  MoveL (T3096) to (114.66, 105.74, 4.1) mm, rotated rx 180 ry 0 rz -180 deg; joints [0, 0, 0, 0, 0, 0]
  Call Extruder 0.46589
  MoveL (T3097) to (103.84, 116.55, 4.1) mm, rotated rx 180 ry 0 rz -180 deg; joints [0, 0, 0, 0, 0, 0]
  Call Extruder 0.07441
  MoveL (T3098) to (103.84, 114.11, 4.1) mm, rotated rx 180 ry 0 rz -180 deg; joints [0, 0, 0, 0, 0, 0]
  Set speed (45.0 mm/s)
  Call Extruder -1.6
  MoveL (T3099) to (103.84, 114.11, 4.1) mm, rotated rx 180 ry 0 rz -180 deg; joints [0, 0, 0, 0, 0, 0]
  Set speed (120.0 mm/s)
  MoveL (T3100) to (103.84, 114.11, 4.1) mm, rotated rx 180 ry 0 rz -180 deg; joints [0, 0, 0, 0, 0, 0]
  Call Extruder -0.38
  MoveL (T3101) to (103.84, 115.17, 4.1) mm, rotated rx 180 ry 0 rz -180 deg; joints [0, 0, 0, 0, 0, 0]
  Set speed (45.0 mm/s)
  Call Extruder -0.02
  MoveL (T3102) to (103.84, 115.17, 4.1) mm, rotated rx 180 ry 0 rz -180 deg; joints [0, 0, 0, 0, 0, 0]
  Set speed (150.0 mm/s)
  MoveL (T3103) to (103.84, 115.17, 6.1) mm, rotated rx 180 ry 0 rz -180 deg; joints [0, 0, 0, 0, 0, 0]
  MoveL (T3104) to (118.71, 121.16, 6.1) mm, rotated rx 180 ry 0 rz -180 deg; joints [0, 0, 0, 0, 0, 0]
  MoveL (T3105) to (118.71, 121.16, 4.1) mm, rotated rx 180 ry 0 rz -180 deg; joints [0, 0, 0, 0, 0, 0]
  Set speed (40.0 mm/s)
  Call Extruder 2.0
  MoveL (T3106) to (118.71, 121.16, 4.1) mm, rotated rx 180 ry 0 rz -180 deg; joints [0, 0, 0, 0, 0, 0]
  Set speed (25.4 mm/s)
  MoveL (T3107) to (118.71, 121.16, 4.1) mm, rotated rx 180 ry 0 rz -180 deg; joints [0, 0, 0, 0, 0, 0]
  Call Extruder 0.07441
  MoveL (T3108) to (121.16, 121.16, 4.1) mm, rotated rx 180 ry 0 rz -180 deg; joints [0, 0, 0, 0, 0, 0]
  Call Extruder 0.7458
  MoveL (T3109) to (103.84, 103.84, 4.1) mm, rotated rx 180 ry 0 rz -180 deg; joints [0, 0, 0, 0, 0, 0]
  Call Extruder 0.07705
  MoveL (T3110) to (106.37, 103.84, 4.1) mm, rotated rx 180 ry 0 rz -180 deg; joints [0, 0, 0, 0, 0, 0]
  Call Extruder 0.02939
  MoveL (T3111) to (106.37, 104.81, 4.1) mm, rotated rx 180 ry 0 rz -180 deg; joints [0, 0, 0, 0, 0, 0]
  Call Extruder 0.10898
  MoveL (T3112) to (103.84, 107.34, 4.1) mm, rotated rx 180 ry 0 rz -180 deg; joints [0, 0, 0, 0, 0, 0]
  Call Extruder 0.03385
  MoveL (T3113) to (103.84, 108.45, 4.1) mm, rotated rx 180 ry 0 rz -180 deg; joints [0, 0, 0, 0, 0, 0]
  Call Extruder 0.54738
  MoveL (T3114) to (116.55, 121.16, 4.1) mm, rotated rx 180 ry 0 rz -180 deg; joints [0, 0, 0, 0, 0, 0]
  Call Extruder 0.03385
  MoveL (T3115) to (117.66, 121.16, 4.1) mm, rotated rx 180 ry 0 rz -180 deg; joints [0, 0, 0, 0, 0, 0]
  Call Extruder 0.15054
  MoveL (T3116) to (121.16, 117.66, 4.1) mm, rotated rx 180 ry 0 rz -180 deg; joints [0, 0, 0, 0, 0, 0]
  Call Extruder 0.03385
  MoveL (T3117) to (121.16, 116.55, 4.1) mm, rotated rx 180 ry 0 rz -180 deg; joints [0, 0, 0, 0, 0, 0]
  Call Extruder 0.46589
  MoveL (T3118) to (110.34, 105.74, 4.1) mm, rotated rx 180 ry 0 rz -180 deg; joints [0, 0, 0, 0, 0, 0]
  Call Extruder 0.0088
  MoveL (T3119) to (110.05, 105.74, 4.1) mm, rotated rx 180 ry 0 rz -180 deg; joints [0, 0, 0, 0, 0, 0]
  Call Extruder 0.26747
  MoveL (T3120) to (103.84, 111.94, 4.1) mm, rotated rx 180 ry 0 rz -180 deg; joints [0, 0, 0, 0, 0, 0]
  Call Extruder 0.03385
  MoveL (T3121) to (103.84, 113.06, 4.1) mm, rotated rx 180 ry 0 rz -180 deg; joints [0, 0, 0, 0, 0, 0]
  Call Extruder 0.34896
  MoveL (T3122) to (111.94, 121.16, 4.1) mm, rotated rx 180 ry 0 rz -180 deg; joints [0, 0, 0, 0, 0, 0]
  Call Extruder 0.03385
  MoveL (T3123) to (113.06, 121.16, 4.1) mm, rotated rx 180 ry 0 rz -180 deg; joints [0, 0, 0, 0, 0, 0]
  Call Extruder 0.29316
  MoveL (T3124) to (119.86, 114.35, 4.1) mm, rotated rx 180 ry 0 rz -180 deg; joints [0, 0, 0, 0, 0, 0]
  Call Extruder 0.03946
  MoveL (T3125) to (121.16, 114.35, 4.1) mm, rotated rx 180 ry 0 rz -180 deg; joints [0, 0, 0, 0, 0, 0]
  Call Extruder 0.03495
  MoveL (T3126) to (121.16, 115.5, 4.1) mm, rotated rx 180 ry 0 rz -180 deg; joints [0, 0, 0, 0, 0, 0]
  Set speed (45.0 mm/s)
  Call Extruder -1.6
  MoveL (T3127) to (121.16, 115.5, 4.1) mm, rotated rx 180 ry 0 rz -180 deg; joints [0, 0, 0, 0, 0, 0]
  Set speed (120.0 mm/s)
  MoveL (T3128) to (121.16, 115.5, 4.1) mm, rotated rx 180 ry 0 rz -180 deg; joints [0, 0, 0, 0, 0, 0]
  Call Extruder -0.38
  MoveL (T3129) to (121.16, 114.43, 4.1) mm, rotated rx 180 ry 0 rz -180 deg; joints [0, 0, 0, 0, 0, 0]
  Set speed (45.0 mm/s)
  Call Extruder -0.02
  MoveL (T3130) to (121.16, 114.43, 4.1) mm, rotated rx 180 ry 0 rz -180 deg; joints [0, 0, 0, 0, 0, 0]
  Set speed (150.0 mm/s)
  MoveL (T3131) to (121.16, 114.43, 6.1) mm, rotated rx 180 ry 0 rz -180 deg; joints [0, 0, 0, 0, 0, 0]
  MoveL (T3132) to (104.34, 103.54, 6.1) mm, rotated rx 180 ry 0 rz -180 deg; joints [0, 0, 0, 0, 0, 0]
  MoveL (T3133) to (104.34, 103.54, 4.3) mm, rotated rx 180 ry 0 rz -180 deg; joints [0, 0, 0, 0, 0, 0]
  Set speed (40.0 mm/s)
  Call Extruder 2.0
  MoveL (T3134) to (104.34, 103.54, 4.3) mm, rotated rx 180 ry 0 rz -180 deg; joints [0, 0, 0, 0, 0, 0]
  Set speed (25.0 mm/s)
  MoveL (T3135) to (104.34, 103.54, 4.3) mm, rotated rx 180 ry 0 rz -180 deg; joints [0, 0, 0, 0, 0, 0]
  Call Extruder 0.07466
  MoveL (T3136) to (106.79, 103.54, 4.3) mm, rotated rx 180 ry 0 rz -180 deg; joints [0, 0, 0, 0, 0, 0]
  Call Extruder 0.05763
  MoveL (T3137) to (106.79, 105.43, 4.3) mm, rotated rx 180 ry 0 rz -180 deg; joints [0, 0, 0, 0, 0, 0]
  Call Extruder 0.11303
  MoveL (T3138) to (110.5, 105.43, 4.3) mm, rotated rx 180 ry 0 rz -180 deg; joints [0, 0, 0, 0, 0, 0]
  Call Extruder 0.05763
  MoveL (T3139) to (110.5, 103.54, 4.3) mm, rotated rx 180 ry 0 rz -180 deg; joints [0, 0, 0, 0, 0, 0]
  Call Extruder 0.09685
  MoveL (T3140) to (113.68, 103.54, 4.3) mm, rotated rx 180 ry 0 rz -180 deg; joints [0, 0, 0, 0, 0, 0]
  Call Extruder 0.05763
  MoveL (T3141) to (113.68, 105.43, 4.3) mm, rotated rx 180 ry 0 rz -180 deg; joints [0, 0, 0, 0, 0, 0]
  Call Extruder 0.11722
  MoveL (T3142) to (117.53, 105.43, 4.3) mm, rotated rx 180 ry 0 rz -180 deg; joints [0, 0, 0, 0, 0, 0]
  Call Extruder 0.05763
  MoveL (T3143) to (117.53, 103.54, 4.3) mm, rotated rx 180 ry 0 rz -180 deg; joints [0, 0, 0, 0, 0, 0]
  Call Extruder 0.11984
  MoveL (T3144) to (121.46, 103.54, 4.3) mm, rotated rx 180 ry 0 rz -180 deg; joints [0, 0, 0, 0, 0, 0]
  Call Extruder 0.2055
  MoveL (T3145) to (121.46, 110.28, 4.3) mm, rotated rx 180 ry 0 rz -180 deg; joints [0, 0, 0, 0, 0, 0]
  Call Extruder 0.05923
  MoveL (T3146) to (119.52, 110.28, 4.3) mm, rotated rx 180 ry 0 rz -180 deg; joints [0, 0, 0, 0, 0, 0]
  Call Extruder 0.11452
  MoveL (T3147) to (119.52, 114.04, 4.3) mm, rotated rx 180 ry 0 rz -180 deg; joints [0, 0, 0, 0, 0, 0]
  Call Extruder 0.05928
  MoveL (T3148) to (121.46, 114.04, 4.3) mm, rotated rx 180 ry 0 rz -180 deg; joints [0, 0, 0, 0, 0, 0]
  Call Extruder 0.22594
  MoveL (T3149) to (121.46, 121.46, 4.3) mm, rotated rx 180 ry 0 rz -180 deg; joints [0, 0, 0, 0, 0, 0]
  Call Extruder 0.54596
  MoveL (T3150) to (103.54, 121.46, 4.3) mm, rotated rx 180 ry 0 rz -180 deg; joints [0, 0, 0, 0, 0, 0]
  Call Extruder 0.54596
  MoveL (T3151) to (103.54, 103.54, 4.3) mm, rotated rx 180 ry 0 rz -180 deg; joints [0, 0, 0, 0, 0, 0]
  Call Extruder 0.02254
  MoveL (T3152) to (104.28, 103.54, 4.3) mm, rotated rx 180 ry 0 rz -180 deg; joints [0, 0, 0, 0, 0, 0]
  Set speed (150.0 mm/s)
  MoveL (T3153) to (103.53, 103.13, 4.3) mm, rotated rx 180 ry 0 rz -180 deg; joints [0, 0, 0, 0, 0, 0]
  Set speed (25.0 mm/s)
  MoveL (T3154) to (103.53, 103.13, 4.3) mm, rotated rx 180 ry 0 rz -180 deg; joints [0, 0, 0, 0, 0, 0]
  Call Extruder 0.11164
  MoveL (T3155) to (107.2, 103.13, 4.3) mm, rotated rx 180 ry 0 rz -180 deg; joints [0, 0, 0, 0, 0, 0]
  Call Extruder 0.05763
  MoveL (T3156) to (107.2, 105.02, 4.3) mm, rotated rx 180 ry 0 rz -180 deg; joints [0, 0, 0, 0, 0, 0]
  Call Extruder 0.08823
  MoveL (T3157) to (110.09, 105.02, 4.3) mm, rotated rx 180 ry 0 rz -180 deg; joints [0, 0, 0, 0, 0, 0]
  Call Extruder 0.05763
  MoveL (T3158) to (110.09, 103.13, 4.3) mm, rotated rx 180 ry 0 rz -180 deg; joints [0, 0, 0, 0, 0, 0]
  Call Extruder 0.12167
  MoveL (T3159) to (114.09, 103.13, 4.3) mm, rotated rx 180 ry 0 rz -180 deg; joints [0, 0, 0, 0, 0, 0]
  Call Extruder 0.05763
  MoveL (T3160) to (114.09, 105.02, 4.3) mm, rotated rx 180 ry 0 rz -180 deg; joints [0, 0, 0, 0, 0, 0]
  Call Extruder 0.09242
  MoveL (T3161) to (117.12, 105.02, 4.3) mm, rotated rx 180 ry 0 rz -180 deg; joints [0, 0, 0, 0, 0, 0]
  Call Extruder 0.05763
  MoveL (T3162) to (117.12, 103.13, 4.3) mm, rotated rx 180 ry 0 rz -180 deg; joints [0, 0, 0, 0, 0, 0]
  Call Extruder 0.14463
  MoveL (T3163) to (121.87, 103.13, 4.3) mm, rotated rx 180 ry 0 rz -180 deg; joints [0, 0, 0, 0, 0, 0]
  Call Extruder 0.23031
  MoveL (T3164) to (121.87, 110.69, 4.3) mm, rotated rx 180 ry 0 rz -180 deg; joints [0, 0, 0, 0, 0, 0]
  Call Extruder 0.05924
  MoveL (T3165) to (119.92, 110.69, 4.3) mm, rotated rx 180 ry 0 rz -180 deg; joints [0, 0, 0, 0, 0, 0]
  Call Extruder 0.08971
  MoveL (T3166) to (119.92, 113.64, 4.3) mm, rotated rx 180 ry 0 rz -180 deg; joints [0, 0, 0, 0, 0, 0]
  Call Extruder 0.05927
  MoveL (T3167) to (121.87, 113.64, 4.3) mm, rotated rx 180 ry 0 rz -180 deg; joints [0, 0, 0, 0, 0, 0]
  Call Extruder 0.25074
  MoveL (T3168) to (121.87, 121.87, 4.3) mm, rotated rx 180 ry 0 rz -180 deg; joints [0, 0, 0, 0, 0, 0]
  Call Extruder 0.57077
  MoveL (T3169) to (103.13, 121.87, 4.3) mm, rotated rx 180 ry 0 rz -180 deg; joints [0, 0, 0, 0, 0, 0]
  Call Extruder 0.57077
  MoveL (T3170) to (103.13, 103.13, 4.3) mm, rotated rx 180 ry 0 rz -180 deg; joints [0, 0, 0, 0, 0, 0]
  Call Extruder 0.01036
  MoveL (T3171) to (103.47, 103.13, 4.3) mm, rotated rx 180 ry 0 rz -180 deg; joints [0, 0, 0, 0, 0, 0]
  Set speed (150.0 mm/s)
  MoveL (T3172) to (102.72, 102.81, 4.3) mm, rotated rx 180 ry 0 rz -180 deg; joints [0, 0, 0, 0, 0, 0]
  Set speed (25.0 mm/s)
  MoveL (T3173) to (102.72, 102.81, 4.3) mm, rotated rx 180 ry 0 rz -180 deg; joints [0, 0, 0, 0, 0, 0]
  Call Extruder 0.00259
  MoveL (T3174) to (102.72, 102.72, 4.3) mm, rotated rx 180 ry 0 rz -180 deg; joints [0, 0, 0, 0, 0, 0]
  Call Extruder 0.14862
  MoveL (T3175) to (107.6, 102.72, 4.3) mm, rotated rx 180 ry 0 rz -180 deg; joints [0, 0, 0, 0, 0, 0]
  Call Extruder 0.05763
  MoveL (T3176) to (107.61, 104.62, 4.3) mm, rotated rx 180 ry 0 rz -180 deg; joints [0, 0, 0, 0, 0, 0]
  Call Extruder 0.06342
  MoveL (T3177) to (109.69, 104.62, 4.3) mm, rotated rx 180 ry 0 rz -180 deg; joints [0, 0, 0, 0, 0, 0]
  Call Extruder 0.05763
  MoveL (T3178) to (109.69, 102.72, 4.3) mm, rotated rx 180 ry 0 rz -180 deg; joints [0, 0, 0, 0, 0, 0]
  Call Extruder 0.14648
  MoveL (T3179) to (114.49, 102.72, 4.3) mm, rotated rx 180 ry 0 rz -180 deg; joints [0, 0, 0, 0, 0, 0]
  Call Extruder 0.05763
  MoveL (T3180) to (114.49, 104.62, 4.3) mm, rotated rx 180 ry 0 rz -180 deg; joints [0, 0, 0, 0, 0, 0]
  Call Extruder 0.06761
  MoveL (T3181) to (116.71, 104.62, 4.3) mm, rotated rx 180 ry 0 rz -180 deg; joints [0, 0, 0, 0, 0, 0]
  Call Extruder 0.05763
  MoveL (T3182) to (116.71, 102.72, 4.3) mm, rotated rx 180 ry 0 rz -180 deg; joints [0, 0, 0, 0, 0, 0]
  Call Extruder 0.16943
  MoveL (T3183) to (122.28, 102.72, 4.3) mm, rotated rx 180 ry 0 rz -180 deg; joints [0, 0, 0, 0, 0, 0]
  Call Extruder 0.25512
  MoveL (T3184) to (122.28, 111.1, 4.3) mm, rotated rx 180 ry 0 rz -180 deg; joints [0, 0, 0, 0, 0, 0]
  Call Extruder 0.05924
  MoveL (T3185) to (120.33, 111.1, 4.3) mm, rotated rx 180 ry 0 rz -180 deg; joints [0, 0, 0, 0, 0, 0]
  Call Extruder 0.06491
  MoveL (T3186) to (120.33, 113.23, 4.3) mm, rotated rx 180 ry 0 rz -180 deg; joints [0, 0, 0, 0, 0, 0]
  Call Extruder 0.05927
  MoveL (T3187) to (122.28, 113.23, 4.3) mm, rotated rx 180 ry 0 rz -180 deg; joints [0, 0, 0, 0, 0, 0]
  Call Extruder 0.27554
  MoveL (T3188) to (122.28, 122.28, 4.3) mm, rotated rx 180 ry 0 rz -180 deg; joints [0, 0, 0, 0, 0, 0]
  Call Extruder 0.59557
  MoveL (T3189) to (102.72, 122.28, 4.3) mm, rotated rx 180 ry 0 rz -180 deg; joints [0, 0, 0, 0, 0, 0]
  Call Extruder 0.59115
  MoveL (T3190) to (102.72, 102.87, 4.3) mm, rotated rx 180 ry 0 rz -180 deg; joints [0, 0, 0, 0, 0, 0]
  Set speed (150.0 mm/s)
  MoveL (T3191) to (102.78, 102.75, 4.3) mm, rotated rx 180 ry 0 rz -180 deg; joints [0, 0, 0, 0, 0, 0]
  Set speed (45.0 mm/s)
  Call Extruder -1.6
  MoveL (T3192) to (102.78, 102.75, 4.3) mm, rotated rx 180 ry 0 rz -180 deg; joints [0, 0, 0, 0, 0, 0]
  Set speed (120.0 mm/s)
  MoveL (T3193) to (102.78, 102.75, 4.3) mm, rotated rx 180 ry 0 rz -180 deg; joints [0, 0, 0, 0, 0, 0]
  Call Extruder -0.05166
  MoveL (T3194) to (102.72, 102.72, 4.3) mm, rotated rx 180 ry 0 rz -180 deg; joints [0, 0, 0, 0, 0, 0]
  Call Extruder -0.32834
  MoveL (T3195) to (103.65, 102.72, 4.3) mm, rotated rx 180 ry 0 rz -180 deg; joints [0, 0, 0, 0, 0, 0]
  Set speed (45.0 mm/s)
  Call Extruder -0.02
  MoveL (T3196) to (103.65, 102.72, 4.3) mm, rotated rx 180 ry 0 rz -180 deg; joints [0, 0, 0, 0, 0, 0]
  Set speed (150.0 mm/s)
  MoveL (T3197) to (103.65, 102.72, 6.3) mm, rotated rx 180 ry 0 rz -180 deg; joints [0, 0, 0, 0, 0, 0]
  MoveL (T3198) to (111.05, 103.66, 6.3) mm, rotated rx 180 ry 0 rz -180 deg; joints [0, 0, 0, 0, 0, 0]
  MoveL (T3199) to (111.05, 103.66, 4.3) mm, rotated rx 180 ry 0 rz -180 deg; joints [0, 0, 0, 0, 0, 0]
  Set speed (40.0 mm/s)
  Call Extruder 2.0
  MoveL (T3200) to (111.05, 103.66, 4.3) mm, rotated rx 180 ry 0 rz -180 deg; joints [0, 0, 0, 0, 0, 0]
  Set speed (25.0 mm/s)
  MoveL (T3201) to (111.05, 103.66, 4.3) mm, rotated rx 180 ry 0 rz -180 deg; joints [0, 0, 0, 0, 0, 0]
  Call Extruder 0.00953
  MoveL (T3202) to (111.24, 103.85, 4.3) mm, rotated rx 180 ry 0 rz -180 deg; joints [0, 0, 0, 0, 0, 0]
  Call Extruder 0.0244
  MoveL (T3203) to (111.24, 104.53, 4.3) mm, rotated rx 180 ry 0 rz -180 deg; joints [0, 0, 0, 0, 0, 0]
  Call Extruder 0.02196
  MoveL (T3204) to (110.81, 104.1, 4.3) mm, rotated rx 180 ry 0 rz -180 deg; joints [0, 0, 0, 0, 0, 0]
  Call Extruder 0.0244
  MoveL (T3205) to (110.81, 104.78, 4.3) mm, rotated rx 180 ry 0 rz -180 deg; joints [0, 0, 0, 0, 0, 0]
  Call Extruder 0.02196
  MoveL (T3206) to (111.24, 105.21, 4.3) mm, rotated rx 180 ry 0 rz -180 deg; joints [0, 0, 0, 0, 0, 0]
  Call Extruder 0.00611
  MoveL (T3207) to (111.24, 105.38, 4.3) mm, rotated rx 180 ry 0 rz -180 deg; joints [0, 0, 0, 0, 0, 0]
  Call Extruder 0.00412
  MoveL (T3208) to (111.16, 105.46, 4.3) mm, rotated rx 180 ry 0 rz -180 deg; joints [0, 0, 0, 0, 0, 0]
  Call Extruder 0.01245
  MoveL (T3209) to (110.81, 105.46, 4.3) mm, rotated rx 180 ry 0 rz -180 deg; joints [0, 0, 0, 0, 0, 0]
  Call Extruder 0.00953
  MoveL (T3210) to (110.62, 105.27, 4.3) mm, rotated rx 180 ry 0 rz -180 deg; joints [0, 0, 0, 0, 0, 0]
  Set speed (150.0 mm/s)
  MoveL (T3211) to (110.74, 105.86, 4.3) mm, rotated rx 180 ry 0 rz -180 deg; joints [0, 0, 0, 0, 0, 0]
  Set speed (25.0 mm/s)
  MoveL (T3212) to (110.74, 105.86, 4.3) mm, rotated rx 180 ry 0 rz -180 deg; joints [0, 0, 0, 0, 0, 0]
  Call Extruder 0.01793
  MoveL (T3213) to (111.33, 105.86, 4.3) mm, rotated rx 180 ry 0 rz -180 deg; joints [0, 0, 0, 0, 0, 0]
  Call Extruder 0.01377
  MoveL (T3214) to (111.65, 105.55, 4.3) mm, rotated rx 180 ry 0 rz -180 deg; joints [0, 0, 0, 0, 0, 0]
  Call Extruder 0.0427
  MoveL (T3215) to (111.64, 104.14, 4.3) mm, rotated rx 180 ry 0 rz -180 deg; joints [0, 0, 0, 0, 0, 0]
  Call Extruder 0.0129
  MoveL (T3216) to (111.94, 103.84, 4.3) mm, rotated rx 180 ry 0 rz -180 deg; joints [0, 0, 0, 0, 0, 0]
  Call Extruder 0.01737
  MoveL (T3217) to (112.52, 103.84, 4.3) mm, rotated rx 180 ry 0 rz -180 deg; joints [0, 0, 0, 0, 0, 0]
  Call Extruder 0.05183
  MoveL (T3218) to (112.51, 105.55, 4.3) mm, rotated rx 180 ry 0 rz -180 deg; joints [0, 0, 0, 0, 0, 0]
  Call Extruder 0.00521
  MoveL (T3219) to (112.64, 105.67, 4.3) mm, rotated rx 180 ry 0 rz -180 deg; joints [0, 0, 0, 0, 0, 0]
  Set speed (150.0 mm/s)
  MoveL (T3220) to (112.74, 103.81, 4.3) mm, rotated rx 180 ry 0 rz -180 deg; joints [0, 0, 0, 0, 0, 0]
  Set speed (25.0 mm/s)
  MoveL (T3221) to (112.74, 103.81, 4.3) mm, rotated rx 180 ry 0 rz -180 deg; joints [0, 0, 0, 0, 0, 0]
  Call Extruder 0.03185
  MoveL (T3222) to (113.37, 104.44, 4.3) mm, rotated rx 180 ry 0 rz -180 deg; joints [0, 0, 0, 0, 0, 0]
  Call Extruder 0.02376
  MoveL (T3223) to (113.37, 105.11, 4.3) mm, rotated rx 180 ry 0 rz -180 deg; joints [0, 0, 0, 0, 0, 0]
  Call Extruder 0.02267
  MoveL (T3224) to (112.92, 104.66, 4.3) mm, rotated rx 180 ry 0 rz -180 deg; joints [0, 0, 0, 0, 0, 0]
  Call Extruder 0.02376
  MoveL (T3225) to (112.92, 105.33, 4.3) mm, rotated rx 180 ry 0 rz -180 deg; joints [0, 0, 0, 0, 0, 0]
  Call Extruder 0.01562
  MoveL (T3226) to (113.23, 105.64, 4.3) mm, rotated rx 180 ry 0 rz -180 deg; joints [0, 0, 0, 0, 0, 0]
  Set speed (45.0 mm/s)
  Call Extruder -1.6
  MoveL (T3227) to (113.23, 105.64, 4.3) mm, rotated rx 180 ry 0 rz -180 deg; joints [0, 0, 0, 0, 0, 0]
  Set speed (120.0 mm/s)
  MoveL (T3228) to (113.23, 105.64, 4.3) mm, rotated rx 180 ry 0 rz -180 deg; joints [0, 0, 0, 0, 0, 0]
  Call Extruder -0.15689
  MoveL (T3229) to (112.92, 105.33, 4.3) mm, rotated rx 180 ry 0 rz -180 deg; joints [0, 0, 0, 0, 0, 0]
  Call Extruder -0.22311
  MoveL (T3230) to (112.92, 104.7, 4.3) mm, rotated rx 180 ry 0 rz -180 deg; joints [0, 0, 0, 0, 0, 0]
  Set speed (45.0 mm/s)
  Call Extruder -0.02
  MoveL (T3231) to (112.92, 104.7, 4.3) mm, rotated rx 180 ry 0 rz -180 deg; joints [0, 0, 0, 0, 0, 0]
  Set speed (150.0 mm/s)
  MoveL (T3232) to (112.92, 104.7, 6.3) mm, rotated rx 180 ry 0 rz -180 deg; joints [0, 0, 0, 0, 0, 0]
  MoveL (T3233) to (121.16, 109.07, 6.3) mm, rotated rx 180 ry 0 rz -180 deg; joints [0, 0, 0, 0, 0, 0]
  MoveL (T3234) to (121.16, 109.07, 4.3) mm, rotated rx 180 ry 0 rz -180 deg; joints [0, 0, 0, 0, 0, 0]
  Set speed (40.0 mm/s)
  Call Extruder 2.0
  MoveL (T3235) to (121.16, 109.07, 4.3) mm, rotated rx 180 ry 0 rz -180 deg; joints [0, 0, 0, 0, 0, 0]
  Set speed (25.0 mm/s)
  MoveL (T3236) to (121.16, 109.07, 4.3) mm, rotated rx 180 ry 0 rz -180 deg; joints [0, 0, 0, 0, 0, 0]
  Call Extruder 0.02783
  MoveL (T3237) to (121.16, 109.98, 4.3) mm, rotated rx 180 ry 0 rz -180 deg; joints [0, 0, 0, 0, 0, 0]
  Call Extruder 0.04657
  MoveL (T3238) to (119.63, 109.98, 4.3) mm, rotated rx 180 ry 0 rz -180 deg; joints [0, 0, 0, 0, 0, 0]
  Call Extruder 0.06587
  MoveL (T3239) to (121.16, 108.45, 4.3) mm, rotated rx 180 ry 0 rz -180 deg; joints [0, 0, 0, 0, 0, 0]
  Call Extruder 0.03385
  MoveL (T3240) to (121.16, 107.34, 4.3) mm, rotated rx 180 ry 0 rz -180 deg; joints [0, 0, 0, 0, 0, 0]
  Call Extruder 0.14318
  MoveL (T3241) to (117.83, 104.02, 4.3) mm, rotated rx 180 ry 0 rz -180 deg; joints [0, 0, 0, 0, 0, 0]
  Call Extruder 0.00521
  MoveL (T3242) to (117.83, 103.84, 4.3) mm, rotated rx 180 ry 0 rz -180 deg; joints [0, 0, 0, 0, 0, 0]
  Call Extruder 0.10124
  MoveL (T3243) to (121.16, 103.84, 4.3) mm, rotated rx 180 ry 0 rz -180 deg; joints [0, 0, 0, 0, 0, 0]
  Call Extruder 0.7458
  MoveL (T3244) to (103.84, 121.16, 4.3) mm, rotated rx 180 ry 0 rz -180 deg; joints [0, 0, 0, 0, 0, 0]
  Call Extruder 0.10645
  MoveL (T3245) to (103.84, 117.66, 4.3) mm, rotated rx 180 ry 0 rz -180 deg; joints [0, 0, 0, 0, 0, 0]
  Call Extruder 0.15054
  MoveL (T3246) to (107.34, 121.16, 4.3) mm, rotated rx 180 ry 0 rz -180 deg; joints [0, 0, 0, 0, 0, 0]
  Call Extruder 0.03385
  MoveL (T3247) to (108.45, 121.16, 4.3) mm, rotated rx 180 ry 0 rz -180 deg; joints [0, 0, 0, 0, 0, 0]
  Call Extruder 0.46362
  MoveL (T3248) to (119.21, 110.39, 4.3) mm, rotated rx 180 ry 0 rz -180 deg; joints [0, 0, 0, 0, 0, 0]
  Call Extruder 0.01201
  MoveL (T3249) to (119.21, 110, 4.3) mm, rotated rx 180 ry 0 rz -180 deg; joints [0, 0, 0, 0, 0, 0]
  Call Extruder 0.1837
  MoveL (T3250) to (114.95, 105.74, 4.3) mm, rotated rx 180 ry 0 rz -180 deg; joints [0, 0, 0, 0, 0, 0]
  Call Extruder 0.00881
  MoveL (T3251) to (114.66, 105.74, 4.3) mm, rotated rx 180 ry 0 rz -180 deg; joints [0, 0, 0, 0, 0, 0]
  Call Extruder 0.46588
  MoveL (T3252) to (103.84, 116.55, 4.3) mm, rotated rx 180 ry 0 rz -180 deg; joints [0, 0, 0, 0, 0, 0]
  Call Extruder 0.07441
  MoveL (T3253) to (103.84, 114.11, 4.3) mm, rotated rx 180 ry 0 rz -180 deg; joints [0, 0, 0, 0, 0, 0]
  Set speed (45.0 mm/s)
  Call Extruder -1.6
  MoveL (T3254) to (103.84, 114.11, 4.3) mm, rotated rx 180 ry 0 rz -180 deg; joints [0, 0, 0, 0, 0, 0]
  Set speed (120.0 mm/s)
  MoveL (T3255) to (103.84, 114.11, 4.3) mm, rotated rx 180 ry 0 rz -180 deg; joints [0, 0, 0, 0, 0, 0]
  Call Extruder -0.38
  MoveL (T3256) to (103.84, 115.17, 4.3) mm, rotated rx 180 ry 0 rz -180 deg; joints [0, 0, 0, 0, 0, 0]
  Set speed (45.0 mm/s)
  Call Extruder -0.02
  MoveL (T3257) to (103.84, 115.17, 4.3) mm, rotated rx 180 ry 0 rz -180 deg; joints [0, 0, 0, 0, 0, 0]
  Set speed (150.0 mm/s)
  MoveL (T3258) to (103.84, 115.17, 6.3) mm, rotated rx 180 ry 0 rz -180 deg; joints [0, 0, 0, 0, 0, 0]
  MoveL (T3259) to (118.71, 121.16, 6.3) mm, rotated rx 180 ry 0 rz -180 deg; joints [0, 0, 0, 0, 0, 0]
  MoveL (T3260) to (118.71, 121.16, 4.3) mm, rotated rx 180 ry 0 rz -180 deg; joints [0, 0, 0, 0, 0, 0]
  Set speed (40.0 mm/s)
  Call Extruder 2.0
  MoveL (T3261) to (118.71, 121.16, 4.3) mm, rotated rx 180 ry 0 rz -180 deg; joints [0, 0, 0, 0, 0, 0]
  Set speed (25.0 mm/s)
  MoveL (T3262) to (118.71, 121.16, 4.3) mm, rotated rx 180 ry 0 rz -180 deg; joints [0, 0, 0, 0, 0, 0]
  Call Extruder 0.07441
  MoveL (T3263) to (121.16, 121.16, 4.3) mm, rotated rx 180 ry 0 rz -180 deg; joints [0, 0, 0, 0, 0, 0]
  Call Extruder 0.7458
  MoveL (T3264) to (103.84, 103.84, 4.3) mm, rotated rx 180 ry 0 rz -180 deg; joints [0, 0, 0, 0, 0, 0]
  Call Extruder 0.08043
  MoveL (T3265) to (106.48, 103.84, 4.3) mm, rotated rx 180 ry 0 rz -180 deg; joints [0, 0, 0, 0, 0, 0]
  Call Extruder 0.02601
  MoveL (T3266) to (106.48, 104.7, 4.3) mm, rotated rx 180 ry 0 rz -180 deg; joints [0, 0, 0, 0, 0, 0]
  Call Extruder 0.11376
  MoveL (T3267) to (103.84, 107.34, 4.3) mm, rotated rx 180 ry 0 rz -180 deg; joints [0, 0, 0, 0, 0, 0]
  Call Extruder 0.03385
  MoveL (T3268) to (103.84, 108.45, 4.3) mm, rotated rx 180 ry 0 rz -180 deg; joints [0, 0, 0, 0, 0, 0]
  Call Extruder 0.54738
  MoveL (T3269) to (116.55, 121.16, 4.3) mm, rotated rx 180 ry 0 rz -180 deg; joints [0, 0, 0, 0, 0, 0]
  Call Extruder 0.03385
  MoveL (T3270) to (117.66, 121.16, 4.3) mm, rotated rx 180 ry 0 rz -180 deg; joints [0, 0, 0, 0, 0, 0]
  Call Extruder 0.15054
  MoveL (T3271) to (121.16, 117.66, 4.3) mm, rotated rx 180 ry 0 rz -180 deg; joints [0, 0, 0, 0, 0, 0]
  Call Extruder 0.03385
  MoveL (T3272) to (121.16, 116.55, 4.3) mm, rotated rx 180 ry 0 rz -180 deg; joints [0, 0, 0, 0, 0, 0]
  Call Extruder 0.46588
  MoveL (T3273) to (110.34, 105.74, 4.3) mm, rotated rx 180 ry 0 rz -180 deg; joints [0, 0, 0, 0, 0, 0]
  Call Extruder 0.00881
  MoveL (T3274) to (110.05, 105.74, 4.3) mm, rotated rx 180 ry 0 rz -180 deg; joints [0, 0, 0, 0, 0, 0]
  Call Extruder 0.26746
  MoveL (T3275) to (103.84, 111.94, 4.3) mm, rotated rx 180 ry 0 rz -180 deg; joints [0, 0, 0, 0, 0, 0]
  Call Extruder 0.03385
  MoveL (T3276) to (103.84, 113.06, 4.3) mm, rotated rx 180 ry 0 rz -180 deg; joints [0, 0, 0, 0, 0, 0]
  Call Extruder 0.34896
  MoveL (T3277) to (111.94, 121.16, 4.3) mm, rotated rx 180 ry 0 rz -180 deg; joints [0, 0, 0, 0, 0, 0]
  Call Extruder 0.03385
  MoveL (T3278) to (113.06, 121.16, 4.3) mm, rotated rx 180 ry 0 rz -180 deg; joints [0, 0, 0, 0, 0, 0]
  Call Extruder 0.29326
  MoveL (T3279) to (119.86, 114.35, 4.3) mm, rotated rx 180 ry 0 rz -180 deg; joints [0, 0, 0, 0, 0, 0]
  Call Extruder 0.03939
  MoveL (T3280) to (121.16, 114.35, 4.3) mm, rotated rx 180 ry 0 rz -180 deg; joints [0, 0, 0, 0, 0, 0]
  Call Extruder 0.03502
  MoveL (T3281) to (121.16, 115.5, 4.3) mm, rotated rx 180 ry 0 rz -180 deg; joints [0, 0, 0, 0, 0, 0]
  Set speed (45.0 mm/s)
  Call Extruder -1.6
  MoveL (T3282) to (121.16, 115.5, 4.3) mm, rotated rx 180 ry 0 rz -180 deg; joints [0, 0, 0, 0, 0, 0]
  Set speed (120.0 mm/s)
  MoveL (T3283) to (121.16, 115.5, 4.3) mm, rotated rx 180 ry 0 rz -180 deg; joints [0, 0, 0, 0, 0, 0]
  Call Extruder -0.38
  MoveL (T3284) to (121.16, 114.43, 4.3) mm, rotated rx 180 ry 0 rz -180 deg; joints [0, 0, 0, 0, 0, 0]
  Set speed (45.0 mm/s)
  Call Extruder -0.02
  MoveL (T3285) to (121.16, 114.43, 4.3) mm, rotated rx 180 ry 0 rz -180 deg; joints [0, 0, 0, 0, 0, 0]
  Set speed (150.0 mm/s)
  MoveL (T3286) to (121.16, 114.43, 6.3) mm, rotated rx 180 ry 0 rz -180 deg; joints [0, 0, 0, 0, 0, 0]
  MoveL (T3287) to (104.34, 103.54, 6.3) mm, rotated rx 180 ry 0 rz -180 deg; joints [0, 0, 0, 0, 0, 0]
  MoveL (T3288) to (104.34, 103.54, 4.5) mm, rotated rx 180 ry 0 rz -180 deg; joints [0, 0, 0, 0, 0, 0]
  Set speed (40.0 mm/s)
  Call Extruder 2.0
  MoveL (T3289) to (104.34, 103.54, 4.5) mm, rotated rx 180 ry 0 rz -180 deg; joints [0, 0, 0, 0, 0, 0]
  Set speed (25.4 mm/s)
  MoveL (T3290) to (104.34, 103.54, 4.5) mm, rotated rx 180 ry 0 rz -180 deg; joints [0, 0, 0, 0, 0, 0]
  Call Extruder 0.07804
  MoveL (T3291) to (106.9, 103.54, 4.5) mm, rotated rx 180 ry 0 rz -180 deg; joints [0, 0, 0, 0, 0, 0]
  Call Extruder 0.05764
  MoveL (T3292) to (106.9, 105.43, 4.5) mm, rotated rx 180 ry 0 rz -180 deg; joints [0, 0, 0, 0, 0, 0]
  Call Extruder 0.11326
  MoveL (T3293) to (110.62, 105.43, 4.5) mm, rotated rx 180 ry 0 rz -180 deg; joints [0, 0, 0, 0, 0, 0]
  Call Extruder 0.05764
  MoveL (T3294) to (110.62, 103.54, 4.5) mm, rotated rx 180 ry 0 rz -180 deg; joints [0, 0, 0, 0, 0, 0]
  Call Extruder 0.08953
  MoveL (T3295) to (113.56, 103.54, 4.5) mm, rotated rx 180 ry 0 rz -180 deg; joints [0, 0, 0, 0, 0, 0]
  Call Extruder 0.05764
  MoveL (T3296) to (113.56, 105.43, 4.5) mm, rotated rx 180 ry 0 rz -180 deg; joints [0, 0, 0, 0, 0, 0]
  Call Extruder 0.11708
  MoveL (T3297) to (117.4, 105.43, 4.5) mm, rotated rx 180 ry 0 rz -180 deg; joints [0, 0, 0, 0, 0, 0]
  Call Extruder 0.05764
  MoveL (T3298) to (117.4, 103.54, 4.5) mm, rotated rx 180 ry 0 rz -180 deg; joints [0, 0, 0, 0, 0, 0]
  Call Extruder 0.12369
  MoveL (T3299) to (121.46, 103.54, 4.5) mm, rotated rx 180 ry 0 rz -180 deg; joints [0, 0, 0, 0, 0, 0]
  Call Extruder 0.20544
  MoveL (T3300) to (121.46, 110.28, 4.5) mm, rotated rx 180 ry 0 rz -180 deg; joints [0, 0, 0, 0, 0, 0]
  Call Extruder 0.05922
  MoveL (T3301) to (119.52, 110.28, 4.5) mm, rotated rx 180 ry 0 rz -180 deg; joints [0, 0, 0, 0, 0, 0]
  Call Extruder 0.11452
  MoveL (T3302) to (119.52, 114.04, 4.5) mm, rotated rx 180 ry 0 rz -180 deg; joints [0, 0, 0, 0, 0, 0]
  Call Extruder 0.05927
  MoveL (T3303) to (121.46, 114.04, 4.5) mm, rotated rx 180 ry 0 rz -180 deg; joints [0, 0, 0, 0, 0, 0]
  Call Extruder 0.22601
  MoveL (T3304) to (121.46, 121.46, 4.5) mm, rotated rx 180 ry 0 rz -180 deg; joints [0, 0, 0, 0, 0, 0]
  Call Extruder 0.54596
  MoveL (T3305) to (103.54, 121.46, 4.5) mm, rotated rx 180 ry 0 rz -180 deg; joints [0, 0, 0, 0, 0, 0]
  Call Extruder 0.54596
  MoveL (T3306) to (103.54, 103.54, 4.5) mm, rotated rx 180 ry 0 rz -180 deg; joints [0, 0, 0, 0, 0, 0]
  Call Extruder 0.02254
  MoveL (T3307) to (104.28, 103.54, 4.5) mm, rotated rx 180 ry 0 rz -180 deg; joints [0, 0, 0, 0, 0, 0]
  Set speed (150.0 mm/s)
  MoveL (T3308) to (103.53, 103.13, 4.5) mm, rotated rx 180 ry 0 rz -180 deg; joints [0, 0, 0, 0, 0, 0]
  Set speed (25.4 mm/s)
  MoveL (T3309) to (103.53, 103.13, 4.5) mm, rotated rx 180 ry 0 rz -180 deg; joints [0, 0, 0, 0, 0, 0]
  Call Extruder 0.11502
  MoveL (T3310) to (107.31, 103.13, 4.5) mm, rotated rx 180 ry 0 rz -180 deg; joints [0, 0, 0, 0, 0, 0]
  Call Extruder 0.05764
  MoveL (T3311) to (107.31, 105.02, 4.5) mm, rotated rx 180 ry 0 rz -180 deg; joints [0, 0, 0, 0, 0, 0]
  Call Extruder 0.08845
  MoveL (T3312) to (110.21, 105.02, 4.5) mm, rotated rx 180 ry 0 rz -180 deg; joints [0, 0, 0, 0, 0, 0]
  Call Extruder 0.05764
  MoveL (T3313) to (110.21, 103.13, 4.5) mm, rotated rx 180 ry 0 rz -180 deg; joints [0, 0, 0, 0, 0, 0]
  Call Extruder 0.11435
  MoveL (T3314) to (113.97, 103.13, 4.5) mm, rotated rx 180 ry 0 rz -180 deg; joints [0, 0, 0, 0, 0, 0]
  Call Extruder 0.05764
  MoveL (T3315) to (113.96, 105.02, 4.5) mm, rotated rx 180 ry 0 rz -180 deg; joints [0, 0, 0, 0, 0, 0]
  Call Extruder 0.09228
  MoveL (T3316) to (116.99, 105.02, 4.5) mm, rotated rx 180 ry 0 rz -180 deg; joints [0, 0, 0, 0, 0, 0]
  Call Extruder 0.05764
  MoveL (T3317) to (116.99, 103.13, 4.5) mm, rotated rx 180 ry 0 rz -180 deg; joints [0, 0, 0, 0, 0, 0]
  Call Extruder 0.14848
  MoveL (T3318) to (121.87, 103.13, 4.5) mm, rotated rx 180 ry 0 rz -180 deg; joints [0, 0, 0, 0, 0, 0]
  Call Extruder 0.23025
  MoveL (T3319) to (121.87, 110.69, 4.5) mm, rotated rx 180 ry 0 rz -180 deg; joints [0, 0, 0, 0, 0, 0]
  Call Extruder 0.05923
  MoveL (T3320) to (119.92, 110.69, 4.5) mm, rotated rx 180 ry 0 rz -180 deg; joints [0, 0, 0, 0, 0, 0]
  Call Extruder 0.08971
  MoveL (T3321) to (119.92, 113.63, 4.5) mm, rotated rx 180 ry 0 rz -180 deg; joints [0, 0, 0, 0, 0, 0]
  Call Extruder 0.05927
  MoveL (T3322) to (121.87, 113.64, 4.5) mm, rotated rx 180 ry 0 rz -180 deg; joints [0, 0, 0, 0, 0, 0]
  Call Extruder 0.25081
  MoveL (T3323) to (121.87, 121.87, 4.5) mm, rotated rx 180 ry 0 rz -180 deg; joints [0, 0, 0, 0, 0, 0]
  Call Extruder 0.57077
  MoveL (T3324) to (103.13, 121.87, 4.5) mm, rotated rx 180 ry 0 rz -180 deg; joints [0, 0, 0, 0, 0, 0]
  Call Extruder 0.57077
  MoveL (T3325) to (103.13, 103.13, 4.5) mm, rotated rx 180 ry 0 rz -180 deg; joints [0, 0, 0, 0, 0, 0]
  Call Extruder 0.01036
  MoveL (T3326) to (103.47, 103.13, 4.5) mm, rotated rx 180 ry 0 rz -180 deg; joints [0, 0, 0, 0, 0, 0]
  Set speed (150.0 mm/s)
  MoveL (T3327) to (102.72, 102.81, 4.5) mm, rotated rx 180 ry 0 rz -180 deg; joints [0, 0, 0, 0, 0, 0]
  Set speed (25.0 mm/s)
  MoveL (T3328) to (102.72, 102.81, 4.5) mm, rotated rx 180 ry 0 rz -180 deg; joints [0, 0, 0, 0, 0, 0]
  Call Extruder 0.00259
  MoveL (T3329) to (102.72, 102.72, 4.5) mm, rotated rx 180 ry 0 rz -180 deg; joints [0, 0, 0, 0, 0, 0]
  Call Extruder 0.152
  MoveL (T3330) to (107.72, 102.72, 4.5) mm, rotated rx 180 ry 0 rz -180 deg; joints [0, 0, 0, 0, 0, 0]
  Call Extruder 0.05764
  MoveL (T3331) to (107.72, 104.62, 4.5) mm, rotated rx 180 ry 0 rz -180 deg; joints [0, 0, 0, 0, 0, 0]
  Call Extruder 0.06365
  MoveL (T3332) to (109.81, 104.62, 4.5) mm, rotated rx 180 ry 0 rz -180 deg; joints [0, 0, 0, 0, 0, 0]
  Call Extruder 0.05764
  MoveL (T3333) to (109.8, 102.72, 4.5) mm, rotated rx 180 ry 0 rz -180 deg; joints [0, 0, 0, 0, 0, 0]
  Call Extruder 0.13916
  MoveL (T3334) to (114.37, 102.72, 4.5) mm, rotated rx 180 ry 0 rz -180 deg; joints [0, 0, 0, 0, 0, 0]
  Call Extruder 0.05764
  MoveL (T3335) to (114.37, 104.62, 4.5) mm, rotated rx 180 ry 0 rz -180 deg; joints [0, 0, 0, 0, 0, 0]
  Call Extruder 0.06747
  MoveL (T3336) to (116.59, 104.62, 4.5) mm, rotated rx 180 ry 0 rz -180 deg; joints [0, 0, 0, 0, 0, 0]
  Call Extruder 0.05764
  MoveL (T3337) to (116.59, 102.72, 4.5) mm, rotated rx 180 ry 0 rz -180 deg; joints [0, 0, 0, 0, 0, 0]
  Call Extruder 0.17328
  MoveL (T3338) to (122.28, 102.72, 4.5) mm, rotated rx 180 ry 0 rz -180 deg; joints [0, 0, 0, 0, 0, 0]
  Call Extruder 0.25505
  MoveL (T3339) to (122.28, 111.1, 4.5) mm, rotated rx 180 ry 0 rz -180 deg; joints [0, 0, 0, 0, 0, 0]
  Call Extruder 0.05923
  MoveL (T3340) to (120.33, 111.1, 4.5) mm, rotated rx 180 ry 0 rz -180 deg; joints [0, 0, 0, 0, 0, 0]
  Call Extruder 0.06491
  MoveL (T3341) to (120.33, 113.23, 4.5) mm, rotated rx 180 ry 0 rz -180 deg; joints [0, 0, 0, 0, 0, 0]
  Call Extruder 0.05926
  MoveL (T3342) to (122.28, 113.23, 4.5) mm, rotated rx 180 ry 0 rz -180 deg; joints [0, 0, 0, 0, 0, 0]
  Call Extruder 0.2756
  MoveL (T3343) to (122.28, 122.28, 4.5) mm, rotated rx 180 ry 0 rz -180 deg; joints [0, 0, 0, 0, 0, 0]
  Call Extruder 0.59557
  MoveL (T3344) to (102.72, 122.28, 4.5) mm, rotated rx 180 ry 0 rz -180 deg; joints [0, 0, 0, 0, 0, 0]
  Call Extruder 0.59115
  MoveL (T3345) to (102.72, 102.87, 4.5) mm, rotated rx 180 ry 0 rz -180 deg; joints [0, 0, 0, 0, 0, 0]
  Set speed (150.0 mm/s)
  MoveL (T3346) to (102.78, 102.75, 4.5) mm, rotated rx 180 ry 0 rz -180 deg; joints [0, 0, 0, 0, 0, 0]
  Set speed (45.0 mm/s)
  Call Extruder -1.6
  MoveL (T3347) to (102.78, 102.75, 4.5) mm, rotated rx 180 ry 0 rz -180 deg; joints [0, 0, 0, 0, 0, 0]
  Set speed (120.0 mm/s)
  MoveL (T3348) to (102.78, 102.75, 4.5) mm, rotated rx 180 ry 0 rz -180 deg; joints [0, 0, 0, 0, 0, 0]
  Call Extruder -0.05166
  MoveL (T3349) to (102.72, 102.72, 4.5) mm, rotated rx 180 ry 0 rz -180 deg; joints [0, 0, 0, 0, 0, 0]
  Call Extruder -0.32834
  MoveL (T3350) to (103.65, 102.72, 4.5) mm, rotated rx 180 ry 0 rz -180 deg; joints [0, 0, 0, 0, 0, 0]
  Set speed (45.0 mm/s)
  Call Extruder -0.02
  MoveL (T3351) to (103.65, 102.72, 4.5) mm, rotated rx 180 ry 0 rz -180 deg; joints [0, 0, 0, 0, 0, 0]
  Set speed (150.0 mm/s)
  MoveL (T3352) to (103.65, 102.72, 6.5) mm, rotated rx 180 ry 0 rz -180 deg; joints [0, 0, 0, 0, 0, 0]
  MoveL (T3353) to (111.05, 105.64, 6.5) mm, rotated rx 180 ry 0 rz -180 deg; joints [0, 0, 0, 0, 0, 0]
  MoveL (T3354) to (111.05, 105.64, 4.5) mm, rotated rx 180 ry 0 rz -180 deg; joints [0, 0, 0, 0, 0, 0]
  Set speed (40.0 mm/s)
  Call Extruder 2.0
  MoveL (T3355) to (111.05, 105.64, 4.5) mm, rotated rx 180 ry 0 rz -180 deg; joints [0, 0, 0, 0, 0, 0]
  Set speed (25.4 mm/s)
  MoveL (T3356) to (111.05, 105.64, 4.5) mm, rotated rx 180 ry 0 rz -180 deg; joints [0, 0, 0, 0, 0, 0]
  Call Extruder 0.01539
  MoveL (T3357) to (111.36, 105.33, 4.5) mm, rotated rx 180 ry 0 rz -180 deg; joints [0, 0, 0, 0, 0, 0]
  Call Extruder 0.02341
  MoveL (T3358) to (111.36, 104.67, 4.5) mm, rotated rx 180 ry 0 rz -180 deg; joints [0, 0, 0, 0, 0, 0]
  Call Extruder 0.0215
  MoveL (T3359) to (110.92, 105.1, 4.5) mm, rotated rx 180 ry 0 rz -180 deg; joints [0, 0, 0, 0, 0, 0]
  Call Extruder 0.02341
  MoveL (T3360) to (110.92, 104.44, 4.5) mm, rotated rx 180 ry 0 rz -180 deg; joints [0, 0, 0, 0, 0, 0]
  Call Extruder 0.03062
  MoveL (T3361) to (111.54, 103.82, 4.5) mm, rotated rx 180 ry 0 rz -180 deg; joints [0, 0, 0, 0, 0, 0]
  Set speed (45.0 mm/s)
  Call Extruder -1.6
  MoveL (T3362) to (111.54, 103.82, 4.5) mm, rotated rx 180 ry 0 rz -180 deg; joints [0, 0, 0, 0, 0, 0]
  Set speed (120.0 mm/s)
  MoveL (T3363) to (111.54, 103.82, 4.5) mm, rotated rx 180 ry 0 rz -180 deg; joints [0, 0, 0, 0, 0, 0]
  Call Extruder -0.30984
  MoveL (T3364) to (110.92, 104.44, 4.5) mm, rotated rx 180 ry 0 rz -180 deg; joints [0, 0, 0, 0, 0, 0]
  Call Extruder -0.07016
  MoveL (T3365) to (110.92, 104.63, 4.5) mm, rotated rx 180 ry 0 rz -180 deg; joints [0, 0, 0, 0, 0, 0]
  Set speed (45.0 mm/s)
  Call Extruder -0.02
  MoveL (T3366) to (110.92, 104.63, 4.5) mm, rotated rx 180 ry 0 rz -180 deg; joints [0, 0, 0, 0, 0, 0]
  Set speed (150.0 mm/s)
  MoveL (T3367) to (110.92, 104.63, 6.5) mm, rotated rx 180 ry 0 rz -180 deg; joints [0, 0, 0, 0, 0, 0]
  MoveL (T3368) to (110.97, 105.87, 6.5) mm, rotated rx 180 ry 0 rz -180 deg; joints [0, 0, 0, 0, 0, 0]
  MoveL (T3369) to (110.97, 105.87, 4.5) mm, rotated rx 180 ry 0 rz -180 deg; joints [0, 0, 0, 0, 0, 0]
  Set speed (40.0 mm/s)
  Call Extruder 2.0
  MoveL (T3370) to (110.97, 105.87, 4.5) mm, rotated rx 180 ry 0 rz -180 deg; joints [0, 0, 0, 0, 0, 0]
  Set speed (25.4 mm/s)
  MoveL (T3371) to (110.97, 105.87, 4.5) mm, rotated rx 180 ry 0 rz -180 deg; joints [0, 0, 0, 0, 0, 0]
  Call Extruder 0.01432
  MoveL (T3372) to (111.44, 105.87, 4.5) mm, rotated rx 180 ry 0 rz -180 deg; joints [0, 0, 0, 0, 0, 0]
  Call Extruder 0.01377
  MoveL (T3373) to (111.76, 105.55, 4.5) mm, rotated rx 180 ry 0 rz -180 deg; joints [0, 0, 0, 0, 0, 0]
  Call Extruder 0.04632
  MoveL (T3374) to (111.76, 104.03, 4.5) mm, rotated rx 180 ry 0 rz -180 deg; joints [0, 0, 0, 0, 0, 0]
  Call Extruder 0.0078
  MoveL (T3375) to (111.94, 103.84, 4.5) mm, rotated rx 180 ry 0 rz -180 deg; joints [0, 0, 0, 0, 0, 0]
  Call Extruder 0.01366
  MoveL (T3376) to (112.39, 103.84, 4.5) mm, rotated rx 180 ry 0 rz -180 deg; joints [0, 0, 0, 0, 0, 0]
  Call Extruder 0.05183
  MoveL (T3377) to (112.39, 105.55, 4.5) mm, rotated rx 180 ry 0 rz -180 deg; joints [0, 0, 0, 0, 0, 0]
  Call Extruder 0.00892
  MoveL (T3378) to (112.6, 105.75, 4.5) mm, rotated rx 180 ry 0 rz -180 deg; joints [0, 0, 0, 0, 0, 0]
  Set speed (150.0 mm/s)
  MoveL (T3379) to (113.43, 105.27, 4.5) mm, rotated rx 180 ry 0 rz -180 deg; joints [0, 0, 0, 0, 0, 0]
  Set speed (25.4 mm/s)
  MoveL (T3380) to (113.43, 105.27, 4.5) mm, rotated rx 180 ry 0 rz -180 deg; joints [0, 0, 0, 0, 0, 0]
  Call Extruder 0.00974
  MoveL (T3381) to (113.24, 105.46, 4.5) mm, rotated rx 180 ry 0 rz -180 deg; joints [0, 0, 0, 0, 0, 0]
  Call Extruder 0.01318
  MoveL (T3382) to (112.88, 105.46, 4.5) mm, rotated rx 180 ry 0 rz -180 deg; joints [0, 0, 0, 0, 0, 0]
  Call Extruder 0.00415
  MoveL (T3383) to (112.8, 105.38, 4.5) mm, rotated rx 180 ry 0 rz -180 deg; joints [0, 0, 0, 0, 0, 0]
  Call Extruder 0.00571
  MoveL (T3384) to (112.8, 105.22, 4.5) mm, rotated rx 180 ry 0 rz -180 deg; joints [0, 0, 0, 0, 0, 0]
  Call Extruder 0.02315
  MoveL (T3385) to (113.25, 104.77, 4.5) mm, rotated rx 180 ry 0 rz -180 deg; joints [0, 0, 0, 0, 0, 0]
  Call Extruder 0.02476
  MoveL (T3386) to (113.25, 104.08, 4.5) mm, rotated rx 180 ry 0 rz -180 deg; joints [0, 0, 0, 0, 0, 0]
  Call Extruder 0.02315
  MoveL (T3387) to (112.8, 104.54, 4.5) mm, rotated rx 180 ry 0 rz -180 deg; joints [0, 0, 0, 0, 0, 0]
  Call Extruder 0.02476
  MoveL (T3388) to (112.8, 103.85, 4.5) mm, rotated rx 180 ry 0 rz -180 deg; joints [0, 0, 0, 0, 0, 0]
  Call Extruder 0.00973
  MoveL (T3389) to (112.99, 103.66, 4.5) mm, rotated rx 180 ry 0 rz -180 deg; joints [0, 0, 0, 0, 0, 0]
  Set speed (45.0 mm/s)
  Call Extruder -1.6
  MoveL (T3390) to (112.99, 103.66, 4.5) mm, rotated rx 180 ry 0 rz -180 deg; joints [0, 0, 0, 0, 0, 0]
  Set speed (120.0 mm/s)
  MoveL (T3391) to (112.99, 103.66, 4.5) mm, rotated rx 180 ry 0 rz -180 deg; joints [0, 0, 0, 0, 0, 0]
  Call Extruder -0.09573
  MoveL (T3392) to (112.8, 103.85, 4.5) mm, rotated rx 180 ry 0 rz -180 deg; joints [0, 0, 0, 0, 0, 0]
  Call Extruder -0.24376
  MoveL (T3393) to (112.8, 104.54, 4.5) mm, rotated rx 180 ry 0 rz -180 deg; joints [0, 0, 0, 0, 0, 0]
  Call Extruder -0.0405
  MoveL (T3394) to (112.88, 104.45, 4.5) mm, rotated rx 180 ry 0 rz -180 deg; joints [0, 0, 0, 0, 0, 0]
  Set speed (45.0 mm/s)
  Call Extruder -0.02
  MoveL (T3395) to (112.88, 104.45, 4.5) mm, rotated rx 180 ry 0 rz -180 deg; joints [0, 0, 0, 0, 0, 0]
  Set speed (150.0 mm/s)
  MoveL (T3396) to (112.88, 104.45, 6.5) mm, rotated rx 180 ry 0 rz -180 deg; joints [0, 0, 0, 0, 0, 0]
  MoveL (T3397) to (121.16, 109.06, 6.5) mm, rotated rx 180 ry 0 rz -180 deg; joints [0, 0, 0, 0, 0, 0]
  MoveL (T3398) to (121.16, 109.06, 4.5) mm, rotated rx 180 ry 0 rz -180 deg; joints [0, 0, 0, 0, 0, 0]
  Set speed (40.0 mm/s)
  Call Extruder 2.0
  MoveL (T3399) to (121.16, 109.06, 4.5) mm, rotated rx 180 ry 0 rz -180 deg; joints [0, 0, 0, 0, 0, 0]
  Set speed (25.4 mm/s)
  MoveL (T3400) to (121.16, 109.06, 4.5) mm, rotated rx 180 ry 0 rz -180 deg; joints [0, 0, 0, 0, 0, 0]
  Call Extruder 0.0279
  MoveL (T3401) to (121.16, 109.98, 4.5) mm, rotated rx 180 ry 0 rz -180 deg; joints [0, 0, 0, 0, 0, 0]
  Call Extruder 0.04651
  MoveL (T3402) to (119.63, 109.98, 4.5) mm, rotated rx 180 ry 0 rz -180 deg; joints [0, 0, 0, 0, 0, 0]
  Call Extruder 0.06577
  MoveL (T3403) to (121.16, 108.45, 4.5) mm, rotated rx 180 ry 0 rz -180 deg; joints [0, 0, 0, 0, 0, 0]
  Call Extruder 0.03385
  MoveL (T3404) to (121.16, 107.34, 4.5) mm, rotated rx 180 ry 0 rz -180 deg; joints [0, 0, 0, 0, 0, 0]
  Call Extruder 0.14862
  MoveL (T3405) to (117.71, 103.89, 4.5) mm, rotated rx 180 ry 0 rz -180 deg; joints [0, 0, 0, 0, 0, 0]
  Call Extruder 0.00136
  MoveL (T3406) to (117.71, 103.84, 4.5) mm, rotated rx 180 ry 0 rz -180 deg; joints [0, 0, 0, 0, 0, 0]
  Call Extruder 0.10509
  MoveL (T3407) to (121.16, 103.84, 4.5) mm, rotated rx 180 ry 0 rz -180 deg; joints [0, 0, 0, 0, 0, 0]
  Call Extruder 0.7458
  MoveL (T3408) to (103.84, 121.16, 4.5) mm, rotated rx 180 ry 0 rz -180 deg; joints [0, 0, 0, 0, 0, 0]
  Call Extruder 0.10645
  MoveL (T3409) to (103.84, 117.66, 4.5) mm, rotated rx 180 ry 0 rz -180 deg; joints [0, 0, 0, 0, 0, 0]
  Call Extruder 0.15054
  MoveL (T3410) to (107.34, 121.16, 4.5) mm, rotated rx 180 ry 0 rz -180 deg; joints [0, 0, 0, 0, 0, 0]
  Call Extruder 0.03385
  MoveL (T3411) to (108.45, 121.16, 4.5) mm, rotated rx 180 ry 0 rz -180 deg; joints [0, 0, 0, 0, 0, 0]
  Call Extruder 0.46363
  MoveL (T3412) to (119.21, 110.39, 4.5) mm, rotated rx 180 ry 0 rz -180 deg; joints [0, 0, 0, 0, 0, 0]
  Call Extruder 0.01199
  MoveL (T3413) to (119.21, 110, 4.5) mm, rotated rx 180 ry 0 rz -180 deg; joints [0, 0, 0, 0, 0, 0]
  Call Extruder 0.18371
  MoveL (T3414) to (114.95, 105.74, 4.5) mm, rotated rx 180 ry 0 rz -180 deg; joints [0, 0, 0, 0, 0, 0]
  Call Extruder 0.00882
  MoveL (T3415) to (114.66, 105.74, 4.5) mm, rotated rx 180 ry 0 rz -180 deg; joints [0, 0, 0, 0, 0, 0]
  Call Extruder 0.46587
  MoveL (T3416) to (103.84, 116.55, 4.5) mm, rotated rx 180 ry 0 rz -180 deg; joints [0, 0, 0, 0, 0, 0]
  Call Extruder 0.07441
  MoveL (T3417) to (103.84, 114.11, 4.5) mm, rotated rx 180 ry 0 rz -180 deg; joints [0, 0, 0, 0, 0, 0]
  Set speed (45.0 mm/s)
  Call Extruder -1.6
  MoveL (T3418) to (103.84, 114.11, 4.5) mm, rotated rx 180 ry 0 rz -180 deg; joints [0, 0, 0, 0, 0, 0]
  Set speed (120.0 mm/s)
  MoveL (T3419) to (103.84, 114.11, 4.5) mm, rotated rx 180 ry 0 rz -180 deg; joints [0, 0, 0, 0, 0, 0]
  Call Extruder -0.38
  MoveL (T3420) to (103.84, 115.17, 4.5) mm, rotated rx 180 ry 0 rz -180 deg; joints [0, 0, 0, 0, 0, 0]
  Set speed (45.0 mm/s)
  Call Extruder -0.02
  MoveL (T3421) to (103.84, 115.17, 4.5) mm, rotated rx 180 ry 0 rz -180 deg; joints [0, 0, 0, 0, 0, 0]
  Set speed (150.0 mm/s)
  MoveL (T3422) to (103.84, 115.17, 6.5) mm, rotated rx 180 ry 0 rz -180 deg; joints [0, 0, 0, 0, 0, 0]
  MoveL (T3423) to (118.71, 121.16, 6.5) mm, rotated rx 180 ry 0 rz -180 deg; joints [0, 0, 0, 0, 0, 0]
  MoveL (T3424) to (118.71, 121.16, 4.5) mm, rotated rx 180 ry 0 rz -180 deg; joints [0, 0, 0, 0, 0, 0]
  Set speed (40.0 mm/s)
  Call Extruder 2.0
  MoveL (T3425) to (118.71, 121.16, 4.5) mm, rotated rx 180 ry 0 rz -180 deg; joints [0, 0, 0, 0, 0, 0]
  Set speed (25.4 mm/s)
  MoveL (T3426) to (118.71, 121.16, 4.5) mm, rotated rx 180 ry 0 rz -180 deg; joints [0, 0, 0, 0, 0, 0]
  Call Extruder 0.07441
  MoveL (T3427) to (121.16, 121.16, 4.5) mm, rotated rx 180 ry 0 rz -180 deg; joints [0, 0, 0, 0, 0, 0]
  Call Extruder 0.7458
  MoveL (T3428) to (103.84, 103.84, 4.5) mm, rotated rx 180 ry 0 rz -180 deg; joints [0, 0, 0, 0, 0, 0]
  Call Extruder 0.08381
  MoveL (T3429) to (106.6, 103.84, 4.5) mm, rotated rx 180 ry 0 rz -180 deg; joints [0, 0, 0, 0, 0, 0]
  Call Extruder 0.02263
  MoveL (T3430) to (106.6, 104.59, 4.5) mm, rotated rx 180 ry 0 rz -180 deg; joints [0, 0, 0, 0, 0, 0]
  Call Extruder 0.11854
  MoveL (T3431) to (103.84, 107.34, 4.5) mm, rotated rx 180 ry 0 rz -180 deg; joints [0, 0, 0, 0, 0, 0]
  Call Extruder 0.03385
  MoveL (T3432) to (103.84, 108.45, 4.5) mm, rotated rx 180 ry 0 rz -180 deg; joints [0, 0, 0, 0, 0, 0]
  Call Extruder 0.54738
  MoveL (T3433) to (116.55, 121.16, 4.5) mm, rotated rx 180 ry 0 rz -180 deg; joints [0, 0, 0, 0, 0, 0]
  Call Extruder 0.03385
  MoveL (T3434) to (117.66, 121.16, 4.5) mm, rotated rx 180 ry 0 rz -180 deg; joints [0, 0, 0, 0, 0, 0]
  Call Extruder 0.15054
  MoveL (T3435) to (121.16, 117.66, 4.5) mm, rotated rx 180 ry 0 rz -180 deg; joints [0, 0, 0, 0, 0, 0]
  Call Extruder 0.03385
  MoveL (T3436) to (121.16, 116.55, 4.5) mm, rotated rx 180 ry 0 rz -180 deg; joints [0, 0, 0, 0, 0, 0]
  Call Extruder 0.46587
  MoveL (T3437) to (110.34, 105.74, 4.5) mm, rotated rx 180 ry 0 rz -180 deg; joints [0, 0, 0, 0, 0, 0]
  Call Extruder 0.00882
  MoveL (T3438) to (110.05, 105.74, 4.5) mm, rotated rx 180 ry 0 rz -180 deg; joints [0, 0, 0, 0, 0, 0]
  Call Extruder 0.26745
  MoveL (T3439) to (103.84, 111.94, 4.5) mm, rotated rx 180 ry 0 rz -180 deg; joints [0, 0, 0, 0, 0, 0]
  Call Extruder 0.03385
  MoveL (T3440) to (103.84, 113.06, 4.5) mm, rotated rx 180 ry 0 rz -180 deg; joints [0, 0, 0, 0, 0, 0]
  Call Extruder 0.34896
  MoveL (T3441) to (111.94, 121.16, 4.5) mm, rotated rx 180 ry 0 rz -180 deg; joints [0, 0, 0, 0, 0, 0]
  Call Extruder 0.03385
  MoveL (T3442) to (113.06, 121.16, 4.5) mm, rotated rx 180 ry 0 rz -180 deg; joints [0, 0, 0, 0, 0, 0]
  Call Extruder 0.29335
  MoveL (T3443) to (119.86, 114.35, 4.5) mm, rotated rx 180 ry 0 rz -180 deg; joints [0, 0, 0, 0, 0, 0]
  Call Extruder 0.03933
  MoveL (T3444) to (121.16, 114.35, 4.5) mm, rotated rx 180 ry 0 rz -180 deg; joints [0, 0, 0, 0, 0, 0]
  Call Extruder 0.03508
  MoveL (T3445) to (121.16, 115.5, 4.5) mm, rotated rx 180 ry 0 rz -180 deg; joints [0, 0, 0, 0, 0, 0]
  Set speed (45.0 mm/s)
  Call Extruder -1.6
  MoveL (T3446) to (121.16, 115.5, 4.5) mm, rotated rx 180 ry 0 rz -180 deg; joints [0, 0, 0, 0, 0, 0]
  Set speed (120.0 mm/s)
  MoveL (T3447) to (121.16, 115.5, 4.5) mm, rotated rx 180 ry 0 rz -180 deg; joints [0, 0, 0, 0, 0, 0]
  Call Extruder -0.38
  MoveL (T3448) to (121.16, 114.43, 4.5) mm, rotated rx 180 ry 0 rz -180 deg; joints [0, 0, 0, 0, 0, 0]
  Set speed (45.0 mm/s)
  Call Extruder -0.02
  MoveL (T3449) to (121.16, 114.43, 4.5) mm, rotated rx 180 ry 0 rz -180 deg; joints [0, 0, 0, 0, 0, 0]
  Set speed (150.0 mm/s)
  MoveL (T3450) to (121.16, 114.43, 6.5) mm, rotated rx 180 ry 0 rz -180 deg; joints [0, 0, 0, 0, 0, 0]
  MoveL (T3451) to (104.34, 103.54, 6.5) mm, rotated rx 180 ry 0 rz -180 deg; joints [0, 0, 0, 0, 0, 0]
  MoveL (T3452) to (104.34, 103.54, 4.7) mm, rotated rx 180 ry 0 rz -180 deg; joints [0, 0, 0, 0, 0, 0]
  Set speed (40.0 mm/s)
  Call Extruder 2.0
  MoveL (T3453) to (104.34, 103.54, 4.7) mm, rotated rx 180 ry 0 rz -180 deg; joints [0, 0, 0, 0, 0, 0]
  Set speed (26.7 mm/s)
  MoveL (T3454) to (104.34, 103.54, 4.7) mm, rotated rx 180 ry 0 rz -180 deg; joints [0, 0, 0, 0, 0, 0]
  Call Extruder 0.08142
  MoveL (T3455) to (107.01, 103.54, 4.7) mm, rotated rx 180 ry 0 rz -180 deg; joints [0, 0, 0, 0, 0, 0]
  Call Extruder 0.05764
  MoveL (T3456) to (107.01, 105.43, 4.7) mm, rotated rx 180 ry 0 rz -180 deg; joints [0, 0, 0, 0, 0, 0]
  Call Extruder 0.11348
  MoveL (T3457) to (110.74, 105.43, 4.7) mm, rotated rx 180 ry 0 rz -180 deg; joints [0, 0, 0, 0, 0, 0]
  Call Extruder 0.05764
  MoveL (T3458) to (110.74, 103.54, 4.7) mm, rotated rx 180 ry 0 rz -180 deg; joints [0, 0, 0, 0, 0, 0]
  Call Extruder 0.08221
  MoveL (T3459) to (113.44, 103.54, 4.7) mm, rotated rx 180 ry 0 rz -180 deg; joints [0, 0, 0, 0, 0, 0]
  Call Extruder 0.05764
  MoveL (T3460) to (113.44, 105.43, 4.7) mm, rotated rx 180 ry 0 rz -180 deg; joints [0, 0, 0, 0, 0, 0]
  Call Extruder 0.11694
  MoveL (T3461) to (117.27, 105.43, 4.7) mm, rotated rx 180 ry 0 rz -180 deg; joints [0, 0, 0, 0, 0, 0]
  Call Extruder 0.05764
  MoveL (T3462) to (117.27, 103.54, 4.7) mm, rotated rx 180 ry 0 rz -180 deg; joints [0, 0, 0, 0, 0, 0]
  Call Extruder 0.12754
  MoveL (T3463) to (121.46, 103.54, 4.7) mm, rotated rx 180 ry 0 rz -180 deg; joints [0, 0, 0, 0, 0, 0]
  Call Extruder 0.20537
  MoveL (T3464) to (121.46, 110.28, 4.7) mm, rotated rx 180 ry 0 rz -180 deg; joints [0, 0, 0, 0, 0, 0]
  Call Extruder 0.05921
  MoveL (T3465) to (119.52, 110.28, 4.7) mm, rotated rx 180 ry 0 rz -180 deg; joints [0, 0, 0, 0, 0, 0]
  Call Extruder 0.11452
  MoveL (T3466) to (119.52, 114.04, 4.7) mm, rotated rx 180 ry 0 rz -180 deg; joints [0, 0, 0, 0, 0, 0]
  Call Extruder 0.05926
  MoveL (T3467) to (121.46, 114.04, 4.7) mm, rotated rx 180 ry 0 rz -180 deg; joints [0, 0, 0, 0, 0, 0]
  Call Extruder 0.22608
  MoveL (T3468) to (121.46, 121.46, 4.7) mm, rotated rx 180 ry 0 rz -180 deg; joints [0, 0, 0, 0, 0, 0]
  Call Extruder 0.54596
  MoveL (T3469) to (103.54, 121.46, 4.7) mm, rotated rx 180 ry 0 rz -180 deg; joints [0, 0, 0, 0, 0, 0]
  Call Extruder 0.54596
  MoveL (T3470) to (103.54, 103.54, 4.7) mm, rotated rx 180 ry 0 rz -180 deg; joints [0, 0, 0, 0, 0, 0]
  Call Extruder 0.02254
  MoveL (T3471) to (104.28, 103.54, 4.7) mm, rotated rx 180 ry 0 rz -180 deg; joints [0, 0, 0, 0, 0, 0]
  Set speed (150.0 mm/s)
  MoveL (T3472) to (103.53, 103.13, 4.7) mm, rotated rx 180 ry 0 rz -180 deg; joints [0, 0, 0, 0, 0, 0]
  Set speed (26.7 mm/s)
  MoveL (T3473) to (103.53, 103.13, 4.7) mm, rotated rx 180 ry 0 rz -180 deg; joints [0, 0, 0, 0, 0, 0]
  Call Extruder 0.1184
  MoveL (T3474) to (107.42, 103.13, 4.7) mm, rotated rx 180 ry 0 rz -180 deg; joints [0, 0, 0, 0, 0, 0]
  Call Extruder 0.05764
  MoveL (T3475) to (107.42, 105.02, 4.7) mm, rotated rx 180 ry 0 rz -180 deg; joints [0, 0, 0, 0, 0, 0]
  Call Extruder 0.08868
  MoveL (T3476) to (110.33, 105.02, 4.7) mm, rotated rx 180 ry 0 rz -180 deg; joints [0, 0, 0, 0, 0, 0]
  Call Extruder 0.05764
  MoveL (T3477) to (110.33, 103.13, 4.7) mm, rotated rx 180 ry 0 rz -180 deg; joints [0, 0, 0, 0, 0, 0]
  Call Extruder 0.10702
  MoveL (T3478) to (113.84, 103.13, 4.7) mm, rotated rx 180 ry 0 rz -180 deg; joints [0, 0, 0, 0, 0, 0]
  Call Extruder 0.05764
  MoveL (T3479) to (113.84, 105.02, 4.7) mm, rotated rx 180 ry 0 rz -180 deg; joints [0, 0, 0, 0, 0, 0]
  Call Extruder 0.09214
  MoveL (T3480) to (116.87, 105.02, 4.7) mm, rotated rx 180 ry 0 rz -180 deg; joints [0, 0, 0, 0, 0, 0]
  Call Extruder 0.05764
  MoveL (T3481) to (116.87, 103.13, 4.7) mm, rotated rx 180 ry 0 rz -180 deg; joints [0, 0, 0, 0, 0, 0]
  Call Extruder 0.15234
  MoveL (T3482) to (121.87, 103.13, 4.7) mm, rotated rx 180 ry 0 rz -180 deg; joints [0, 0, 0, 0, 0, 0]
  Call Extruder 0.23018
  MoveL (T3483) to (121.87, 110.69, 4.7) mm, rotated rx 180 ry 0 rz -180 deg; joints [0, 0, 0, 0, 0, 0]
  Call Extruder 0.05922
  MoveL (T3484) to (119.92, 110.69, 4.7) mm, rotated rx 180 ry 0 rz -180 deg; joints [0, 0, 0, 0, 0, 0]
  Call Extruder 0.08971
  MoveL (T3485) to (119.92, 113.63, 4.7) mm, rotated rx 180 ry 0 rz -180 deg; joints [0, 0, 0, 0, 0, 0]
  Call Extruder 0.05926
  MoveL (T3486) to (121.87, 113.63, 4.7) mm, rotated rx 180 ry 0 rz -180 deg; joints [0, 0, 0, 0, 0, 0]
  Call Extruder 0.25087
  MoveL (T3487) to (121.87, 121.87, 4.7) mm, rotated rx 180 ry 0 rz -180 deg; joints [0, 0, 0, 0, 0, 0]
  Call Extruder 0.57077
  MoveL (T3488) to (103.13, 121.87, 4.7) mm, rotated rx 180 ry 0 rz -180 deg; joints [0, 0, 0, 0, 0, 0]
  Call Extruder 0.57077
  MoveL (T3489) to (103.13, 103.13, 4.7) mm, rotated rx 180 ry 0 rz -180 deg; joints [0, 0, 0, 0, 0, 0]
  Call Extruder 0.01036
  MoveL (T3490) to (103.47, 103.13, 4.7) mm, rotated rx 180 ry 0 rz -180 deg; joints [0, 0, 0, 0, 0, 0]
  Set speed (150.0 mm/s)
  MoveL (T3491) to (102.72, 102.81, 4.7) mm, rotated rx 180 ry 0 rz -180 deg; joints [0, 0, 0, 0, 0, 0]
  Set speed (25.0 mm/s)
  MoveL (T3492) to (102.72, 102.81, 4.7) mm, rotated rx 180 ry 0 rz -180 deg; joints [0, 0, 0, 0, 0, 0]
  Call Extruder 0.00259
  MoveL (T3493) to (102.72, 102.72, 4.7) mm, rotated rx 180 ry 0 rz -180 deg; joints [0, 0, 0, 0, 0, 0]
  Call Extruder 0.15539
  MoveL (T3494) to (107.83, 102.72, 4.7) mm, rotated rx 180 ry 0 rz -180 deg; joints [0, 0, 0, 0, 0, 0]
  Call Extruder 0.05764
  MoveL (T3495) to (107.83, 104.62, 4.7) mm, rotated rx 180 ry 0 rz -180 deg; joints [0, 0, 0, 0, 0, 0]
  Call Extruder 0.06388
  MoveL (T3496) to (109.92, 104.62, 4.7) mm, rotated rx 180 ry 0 rz -180 deg; joints [0, 0, 0, 0, 0, 0]
  Call Extruder 0.05764
  MoveL (T3497) to (109.92, 102.72, 4.7) mm, rotated rx 180 ry 0 rz -180 deg; joints [0, 0, 0, 0, 0, 0]
  Call Extruder 0.13184
  MoveL (T3498) to (114.25, 102.72, 4.7) mm, rotated rx 180 ry 0 rz -180 deg; joints [0, 0, 0, 0, 0, 0]
  Call Extruder 0.05764
  MoveL (T3499) to (114.25, 104.62, 4.7) mm, rotated rx 180 ry 0 rz -180 deg; joints [0, 0, 0, 0, 0, 0]
  Call Extruder 0.06733
  MoveL (T3500) to (116.46, 104.62, 4.7) mm, rotated rx 180 ry 0 rz -180 deg; joints [0, 0, 0, 0, 0, 0]
  Call Extruder 0.05764
  MoveL (T3501) to (116.46, 102.72, 4.7) mm, rotated rx 180 ry 0 rz -180 deg; joints [0, 0, 0, 0, 0, 0]
  Call Extruder 0.17713
  MoveL (T3502) to (122.28, 102.72, 4.7) mm, rotated rx 180 ry 0 rz -180 deg; joints [0, 0, 0, 0, 0, 0]
  Call Extruder 0.25499
  MoveL (T3503) to (122.28, 111.09, 4.7) mm, rotated rx 180 ry 0 rz -180 deg; joints [0, 0, 0, 0, 0, 0]
  Call Extruder 0.05922
  MoveL (T3504) to (120.33, 111.09, 4.7) mm, rotated rx 180 ry 0 rz -180 deg; joints [0, 0, 0, 0, 0, 0]
  Call Extruder 0.06491
  MoveL (T3505) to (120.33, 113.22, 4.7) mm, rotated rx 180 ry 0 rz -180 deg; joints [0, 0, 0, 0, 0, 0]
  Call Extruder 0.05925
  MoveL (T3506) to (122.28, 113.23, 4.7) mm, rotated rx 180 ry 0 rz -180 deg; joints [0, 0, 0, 0, 0, 0]
  Call Extruder 0.27567
  MoveL (T3507) to (122.28, 122.28, 4.7) mm, rotated rx 180 ry 0 rz -180 deg; joints [0, 0, 0, 0, 0, 0]
  Call Extruder 0.59557
  MoveL (T3508) to (102.72, 122.28, 4.7) mm, rotated rx 180 ry 0 rz -180 deg; joints [0, 0, 0, 0, 0, 0]
  Call Extruder 0.59115
  MoveL (T3509) to (102.72, 102.87, 4.7) mm, rotated rx 180 ry 0 rz -180 deg; joints [0, 0, 0, 0, 0, 0]
  Set speed (150.0 mm/s)
  MoveL (T3510) to (102.78, 102.75, 4.7) mm, rotated rx 180 ry 0 rz -180 deg; joints [0, 0, 0, 0, 0, 0]
  Set speed (45.0 mm/s)
  Call Extruder -1.6
  MoveL (T3511) to (102.78, 102.75, 4.7) mm, rotated rx 180 ry 0 rz -180 deg; joints [0, 0, 0, 0, 0, 0]
  Set speed (120.0 mm/s)
  MoveL (T3512) to (102.78, 102.75, 4.7) mm, rotated rx 180 ry 0 rz -180 deg; joints [0, 0, 0, 0, 0, 0]
  Call Extruder -0.05166
  MoveL (T3513) to (102.72, 102.72, 4.7) mm, rotated rx 180 ry 0 rz -180 deg; joints [0, 0, 0, 0, 0, 0]
  Call Extruder -0.32834
  MoveL (T3514) to (103.65, 102.72, 4.7) mm, rotated rx 180 ry 0 rz -180 deg; joints [0, 0, 0, 0, 0, 0]
  Set speed (45.0 mm/s)
  Call Extruder -0.02
  MoveL (T3515) to (103.65, 102.72, 4.7) mm, rotated rx 180 ry 0 rz -180 deg; joints [0, 0, 0, 0, 0, 0]
  Set speed (150.0 mm/s)
  MoveL (T3516) to (103.65, 102.72, 6.7) mm, rotated rx 180 ry 0 rz -180 deg; joints [0, 0, 0, 0, 0, 0]
  MoveL (T3517) to (106.36, 103.99, 6.7) mm, rotated rx 180 ry 0 rz -180 deg; joints [0, 0, 0, 0, 0, 0]
  MoveL (T3518) to (106.36, 103.99, 4.7) mm, rotated rx 180 ry 0 rz -180 deg; joints [0, 0, 0, 0, 0, 0]
  Set speed (40.0 mm/s)
  Call Extruder 2.0
  MoveL (T3519) to (106.36, 103.99, 4.7) mm, rotated rx 180 ry 0 rz -180 deg; joints [0, 0, 0, 0, 0, 0]
  Set speed (26.7 mm/s)
  MoveL (T3520) to (106.36, 103.99, 4.7) mm, rotated rx 180 ry 0 rz -180 deg; joints [0, 0, 0, 0, 0, 0]
  Call Extruder 0.0156
  MoveL (T3521) to (106.71, 104.33, 4.7) mm, rotated rx 180 ry 0 rz -180 deg; joints [0, 0, 0, 0, 0, 0]
  Call Extruder 0.01892
  MoveL (T3522) to (106.71, 104.93, 4.7) mm, rotated rx 180 ry 0 rz -180 deg; joints [0, 0, 0, 0, 0, 0]
  Call Extruder 0.0074
  MoveL (T3523) to (106.54, 104.77, 4.7) mm, rotated rx 180 ry 0 rz -180 deg; joints [0, 0, 0, 0, 0, 0]
  Call Extruder 0.01892
  MoveL (T3524) to (106.54, 105.36, 4.7) mm, rotated rx 180 ry 0 rz -180 deg; joints [0, 0, 0, 0, 0, 0]
  Call Extruder 0.01231
  MoveL (T3525) to (106.82, 105.64, 4.7) mm, rotated rx 180 ry 0 rz -180 deg; joints [0, 0, 0, 0, 0, 0]
  Set speed (45.0 mm/s)
  Call Extruder -1.6
  MoveL (T3526) to (106.82, 105.64, 4.7) mm, rotated rx 180 ry 0 rz -180 deg; joints [0, 0, 0, 0, 0, 0]
  Set speed (120.0 mm/s)
  MoveL (T3527) to (106.82, 105.64, 4.7) mm, rotated rx 180 ry 0 rz -180 deg; joints [0, 0, 0, 0, 0, 0]
  Call Extruder -0.13863
  MoveL (T3528) to (106.54, 105.36, 4.7) mm, rotated rx 180 ry 0 rz -180 deg; joints [0, 0, 0, 0, 0, 0]
  Call Extruder -0.21308
  MoveL (T3529) to (106.54, 104.77, 4.7) mm, rotated rx 180 ry 0 rz -180 deg; joints [0, 0, 0, 0, 0, 0]
  Call Extruder -0.02829
  MoveL (T3530) to (106.6, 104.82, 4.7) mm, rotated rx 180 ry 0 rz -180 deg; joints [0, 0, 0, 0, 0, 0]
  Set speed (45.0 mm/s)
  Call Extruder -0.02
  MoveL (T3531) to (106.6, 104.82, 4.7) mm, rotated rx 180 ry 0 rz -180 deg; joints [0, 0, 0, 0, 0, 0]
  Set speed (150.0 mm/s)
  MoveL (T3532) to (106.6, 104.82, 6.7) mm, rotated rx 180 ry 0 rz -180 deg; joints [0, 0, 0, 0, 0, 0]
  MoveL (T3533) to (111.21, 105.87, 6.7) mm, rotated rx 180 ry 0 rz -180 deg; joints [0, 0, 0, 0, 0, 0]
  MoveL (T3534) to (111.21, 105.87, 4.7) mm, rotated rx 180 ry 0 rz -180 deg; joints [0, 0, 0, 0, 0, 0]
  Set speed (40.0 mm/s)
  Call Extruder 2.0
  MoveL (T3535) to (111.21, 105.87, 4.7) mm, rotated rx 180 ry 0 rz -180 deg; joints [0, 0, 0, 0, 0, 0]
  Set speed (26.7 mm/s)
  MoveL (T3536) to (111.21, 105.87, 4.7) mm, rotated rx 180 ry 0 rz -180 deg; joints [0, 0, 0, 0, 0, 0]
  Call Extruder 0.01071
  MoveL (T3537) to (111.56, 105.87, 4.7) mm, rotated rx 180 ry 0 rz -180 deg; joints [0, 0, 0, 0, 0, 0]
  Call Extruder 0.01377
  MoveL (T3538) to (111.88, 105.55, 4.7) mm, rotated rx 180 ry 0 rz -180 deg; joints [0, 0, 0, 0, 0, 0]
  Call Extruder 0.04993
  MoveL (T3539) to (111.88, 103.91, 4.7) mm, rotated rx 180 ry 0 rz -180 deg; joints [0, 0, 0, 0, 0, 0]
  Call Extruder 0.0027
  MoveL (T3540) to (111.94, 103.84, 4.7) mm, rotated rx 180 ry 0 rz -180 deg; joints [0, 0, 0, 0, 0, 0]
  Call Extruder 0.00995
  MoveL (T3541) to (112.27, 103.84, 4.7) mm, rotated rx 180 ry 0 rz -180 deg; joints [0, 0, 0, 0, 0, 0]
  Call Extruder 0.05184
  MoveL (T3542) to (112.27, 105.55, 4.7) mm, rotated rx 180 ry 0 rz -180 deg; joints [0, 0, 0, 0, 0, 0]
  Call Extruder 0.01262
  MoveL (T3543) to (112.56, 105.84, 4.7) mm, rotated rx 180 ry 0 rz -180 deg; joints [0, 0, 0, 0, 0, 0]
  Set speed (45.0 mm/s)
  Call Extruder -1.6
  MoveL (T3544) to (112.56, 105.84, 4.7) mm, rotated rx 180 ry 0 rz -180 deg; joints [0, 0, 0, 0, 0, 0]
  Set speed (120.0 mm/s)
  MoveL (T3545) to (112.56, 105.84, 4.7) mm, rotated rx 180 ry 0 rz -180 deg; joints [0, 0, 0, 0, 0, 0]
  Call Extruder -0.14761
  MoveL (T3546) to (112.27, 105.55, 4.7) mm, rotated rx 180 ry 0 rz -180 deg; joints [0, 0, 0, 0, 0, 0]
  Call Extruder -0.23239
  MoveL (T3547) to (112.27, 104.89, 4.7) mm, rotated rx 180 ry 0 rz -180 deg; joints [0, 0, 0, 0, 0, 0]
  Set speed (45.0 mm/s)
  Call Extruder -0.02
  MoveL (T3548) to (112.27, 104.89, 4.7) mm, rotated rx 180 ry 0 rz -180 deg; joints [0, 0, 0, 0, 0, 0]
  Set speed (150.0 mm/s)
  MoveL (T3549) to (112.27, 104.89, 6.7) mm, rotated rx 180 ry 0 rz -180 deg; joints [0, 0, 0, 0, 0, 0]
  MoveL (T3550) to (112.5, 103.81, 6.7) mm, rotated rx 180 ry 0 rz -180 deg; joints [0, 0, 0, 0, 0, 0]
  MoveL (T3551) to (112.5, 103.81, 4.7) mm, rotated rx 180 ry 0 rz -180 deg; joints [0, 0, 0, 0, 0, 0]
  Set speed (40.0 mm/s)
  Call Extruder 2.0
  MoveL (T3552) to (112.5, 103.81, 4.7) mm, rotated rx 180 ry 0 rz -180 deg; joints [0, 0, 0, 0, 0, 0]
  Set speed (26.7 mm/s)
  MoveL (T3553) to (112.5, 103.81, 4.7) mm, rotated rx 180 ry 0 rz -180 deg; joints [0, 0, 0, 0, 0, 0]
  Call Extruder 0.03186
  MoveL (T3554) to (113.13, 104.44, 4.7) mm, rotated rx 180 ry 0 rz -180 deg; joints [0, 0, 0, 0, 0, 0]
  Call Extruder 0.02376
  MoveL (T3555) to (113.13, 105.11, 4.7) mm, rotated rx 180 ry 0 rz -180 deg; joints [0, 0, 0, 0, 0, 0]
  Call Extruder 0.02267
  MoveL (T3556) to (112.68, 104.66, 4.7) mm, rotated rx 180 ry 0 rz -180 deg; joints [0, 0, 0, 0, 0, 0]
  Call Extruder 0.02376
  MoveL (T3557) to (112.68, 105.33, 4.7) mm, rotated rx 180 ry 0 rz -180 deg; joints [0, 0, 0, 0, 0, 0]
  Call Extruder 0.01562
  MoveL (T3558) to (112.99, 105.64, 4.7) mm, rotated rx 180 ry 0 rz -180 deg; joints [0, 0, 0, 0, 0, 0]
  Set speed (45.0 mm/s)
  Call Extruder -1.6
  MoveL (T3559) to (112.99, 105.64, 4.7) mm, rotated rx 180 ry 0 rz -180 deg; joints [0, 0, 0, 0, 0, 0]
  Set speed (120.0 mm/s)
  MoveL (T3560) to (112.99, 105.64, 4.7) mm, rotated rx 180 ry 0 rz -180 deg; joints [0, 0, 0, 0, 0, 0]
  Call Extruder -0.15692
  MoveL (T3561) to (112.68, 105.33, 4.7) mm, rotated rx 180 ry 0 rz -180 deg; joints [0, 0, 0, 0, 0, 0]
  Call Extruder -0.22308
  MoveL (T3562) to (112.68, 104.7, 4.7) mm, rotated rx 180 ry 0 rz -180 deg; joints [0, 0, 0, 0, 0, 0]
  Set speed (45.0 mm/s)
  Call Extruder -0.02
  MoveL (T3563) to (112.68, 104.7, 4.7) mm, rotated rx 180 ry 0 rz -180 deg; joints [0, 0, 0, 0, 0, 0]
  Set speed (150.0 mm/s)
  MoveL (T3564) to (112.68, 104.7, 6.7) mm, rotated rx 180 ry 0 rz -180 deg; joints [0, 0, 0, 0, 0, 0]
  MoveL (T3565) to (111.29, 103.66, 6.7) mm, rotated rx 180 ry 0 rz -180 deg; joints [0, 0, 0, 0, 0, 0]
  MoveL (T3566) to (111.29, 103.66, 4.7) mm, rotated rx 180 ry 0 rz -180 deg; joints [0, 0, 0, 0, 0, 0]
  Set speed (40.0 mm/s)
  Call Extruder 2.0
  MoveL (T3567) to (111.29, 103.66, 4.7) mm, rotated rx 180 ry 0 rz -180 deg; joints [0, 0, 0, 0, 0, 0]
  Set speed (26.7 mm/s)
  MoveL (T3568) to (111.29, 103.66, 4.7) mm, rotated rx 180 ry 0 rz -180 deg; joints [0, 0, 0, 0, 0, 0]
  Call Extruder 0.00954
  MoveL (T3569) to (111.47, 103.85, 4.7) mm, rotated rx 180 ry 0 rz -180 deg; joints [0, 0, 0, 0, 0, 0]
  Call Extruder 0.0244
  MoveL (T3570) to (111.47, 104.53, 4.7) mm, rotated rx 180 ry 0 rz -180 deg; joints [0, 0, 0, 0, 0, 0]
  Call Extruder 0.02197
  MoveL (T3571) to (111.04, 104.1, 4.7) mm, rotated rx 180 ry 0 rz -180 deg; joints [0, 0, 0, 0, 0, 0]
  Call Extruder 0.0244
  MoveL (T3572) to (111.04, 104.78, 4.7) mm, rotated rx 180 ry 0 rz -180 deg; joints [0, 0, 0, 0, 0, 0]
  Call Extruder 0.02197
  MoveL (T3573) to (111.47, 105.21, 4.7) mm, rotated rx 180 ry 0 rz -180 deg; joints [0, 0, 0, 0, 0, 0]
  Call Extruder 0.00611
  MoveL (T3574) to (111.47, 105.38, 4.7) mm, rotated rx 180 ry 0 rz -180 deg; joints [0, 0, 0, 0, 0, 0]
  Call Extruder 0.00412
  MoveL (T3575) to (111.39, 105.46, 4.7) mm, rotated rx 180 ry 0 rz -180 deg; joints [0, 0, 0, 0, 0, 0]
  Call Extruder 0.01245
  MoveL (T3576) to (111.05, 105.46, 4.7) mm, rotated rx 180 ry 0 rz -180 deg; joints [0, 0, 0, 0, 0, 0]
  Call Extruder 0.00953
  MoveL (T3577) to (110.86, 105.27, 4.7) mm, rotated rx 180 ry 0 rz -180 deg; joints [0, 0, 0, 0, 0, 0]
  Set speed (45.0 mm/s)
  Call Extruder -1.6
  MoveL (T3578) to (110.86, 105.27, 4.7) mm, rotated rx 180 ry 0 rz -180 deg; joints [0, 0, 0, 0, 0, 0]
  Set speed (120.0 mm/s)
  MoveL (T3579) to (110.86, 105.27, 4.7) mm, rotated rx 180 ry 0 rz -180 deg; joints [0, 0, 0, 0, 0, 0]
  Call Extruder -0.09452
  MoveL (T3580) to (111.05, 105.46, 4.7) mm, rotated rx 180 ry 0 rz -180 deg; joints [0, 0, 0, 0, 0, 0]
  Call Extruder -0.1235
  MoveL (T3581) to (111.39, 105.46, 4.7) mm, rotated rx 180 ry 0 rz -180 deg; joints [0, 0, 0, 0, 0, 0]
  Call Extruder -0.04086
  MoveL (T3582) to (111.47, 105.38, 4.7) mm, rotated rx 180 ry 0 rz -180 deg; joints [0, 0, 0, 0, 0, 0]
  Call Extruder -0.06061
  MoveL (T3583) to (111.47, 105.21, 4.7) mm, rotated rx 180 ry 0 rz -180 deg; joints [0, 0, 0, 0, 0, 0]
  Call Extruder -0.06051
  MoveL (T3584) to (111.36, 105.09, 4.7) mm, rotated rx 180 ry 0 rz -180 deg; joints [0, 0, 0, 0, 0, 0]
  Set speed (45.0 mm/s)
  Call Extruder -0.02
  MoveL (T3585) to (111.36, 105.09, 4.7) mm, rotated rx 180 ry 0 rz -180 deg; joints [0, 0, 0, 0, 0, 0]
  Set speed (150.0 mm/s)
  MoveL (T3586) to (111.36, 105.09, 6.7) mm, rotated rx 180 ry 0 rz -180 deg; joints [0, 0, 0, 0, 0, 0]
  MoveL (T3587) to (117.4, 104.04, 6.7) mm, rotated rx 180 ry 0 rz -180 deg; joints [0, 0, 0, 0, 0, 0]
  MoveL (T3588) to (117.4, 104.04, 4.7) mm, rotated rx 180 ry 0 rz -180 deg; joints [0, 0, 0, 0, 0, 0]
  Set speed (40.0 mm/s)
  Call Extruder 2.0
  MoveL (T3589) to (117.4, 104.04, 4.7) mm, rotated rx 180 ry 0 rz -180 deg; joints [0, 0, 0, 0, 0, 0]
  Set speed (26.7 mm/s)
  MoveL (T3590) to (117.4, 104.04, 4.7) mm, rotated rx 180 ry 0 rz -180 deg; joints [0, 0, 0, 0, 0, 0]
  Call Extruder 0.01926
  MoveL (T3591) to (117.81, 104.45, 4.7) mm, rotated rx 180 ry 0 rz -180 deg; joints [0, 0, 0, 0, 0, 0]
  Call Extruder 0.02084
  MoveL (T3592) to (117.81, 105.08, 4.7) mm, rotated rx 180 ry 0 rz -180 deg; joints [0, 0, 0, 0, 0, 0]
  Call Extruder 0.01926
  MoveL (T3593) to (117.4, 104.67, 4.7) mm, rotated rx 180 ry 0 rz -180 deg; joints [0, 0, 0, 0, 0, 0]
  Set speed (45.0 mm/s)
  Call Extruder -1.6
  MoveL (T3594) to (117.4, 104.67, 4.7) mm, rotated rx 180 ry 0 rz -180 deg; joints [0, 0, 0, 0, 0, 0]
  Set speed (120.0 mm/s)
  MoveL (T3595) to (117.4, 104.67, 4.7) mm, rotated rx 180 ry 0 rz -180 deg; joints [0, 0, 0, 0, 0, 0]
  Call Extruder -0.20654
  MoveL (T3596) to (117.81, 105.08, 4.7) mm, rotated rx 180 ry 0 rz -180 deg; joints [0, 0, 0, 0, 0, 0]
  Call Extruder -0.17346
  MoveL (T3597) to (117.81, 104.59, 4.7) mm, rotated rx 180 ry 0 rz -180 deg; joints [0, 0, 0, 0, 0, 0]
  Set speed (45.0 mm/s)
  Call Extruder -0.02
  MoveL (T3598) to (117.81, 104.59, 4.7) mm, rotated rx 180 ry 0 rz -180 deg; joints [0, 0, 0, 0, 0, 0]
  Set speed (150.0 mm/s)
  MoveL (T3599) to (117.81, 104.59, 6.7) mm, rotated rx 180 ry 0 rz -180 deg; joints [0, 0, 0, 0, 0, 0]
  MoveL (T3600) to (121.16, 109.06, 6.7) mm, rotated rx 180 ry 0 rz -180 deg; joints [0, 0, 0, 0, 0, 0]
  MoveL (T3601) to (121.16, 109.06, 4.7) mm, rotated rx 180 ry 0 rz -180 deg; joints [0, 0, 0, 0, 0, 0]
  Set speed (40.0 mm/s)
  Call Extruder 2.0
  MoveL (T3602) to (121.16, 109.06, 4.7) mm, rotated rx 180 ry 0 rz -180 deg; joints [0, 0, 0, 0, 0, 0]
  Set speed (26.7 mm/s)
  MoveL (T3603) to (121.16, 109.06, 4.7) mm, rotated rx 180 ry 0 rz -180 deg; joints [0, 0, 0, 0, 0, 0]
  Call Extruder 0.02796
  MoveL (T3604) to (121.16, 109.97, 4.7) mm, rotated rx 180 ry 0 rz -180 deg; joints [0, 0, 0, 0, 0, 0]
  Call Extruder 0.04644
  MoveL (T3605) to (119.63, 109.97, 4.7) mm, rotated rx 180 ry 0 rz -180 deg; joints [0, 0, 0, 0, 0, 0]
  Call Extruder 0.06568
  MoveL (T3606) to (121.16, 108.45, 4.7) mm, rotated rx 180 ry 0 rz -180 deg; joints [0, 0, 0, 0, 0, 0]
  Call Extruder 0.03385
  MoveL (T3607) to (121.16, 107.34, 4.7) mm, rotated rx 180 ry 0 rz -180 deg; joints [0, 0, 0, 0, 0, 0]
  Call Extruder 0.12677
  MoveL (T3608) to (118.21, 104.4, 4.7) mm, rotated rx 180 ry 0 rz -180 deg; joints [0, 0, 0, 0, 0, 0]
  Call Extruder 0.01681
  MoveL (T3609) to (118.21, 103.84, 4.7) mm, rotated rx 180 ry 0 rz -180 deg; joints [0, 0, 0, 0, 0, 0]
  Call Extruder 0.08963
  MoveL (T3610) to (121.16, 103.84, 4.7) mm, rotated rx 180 ry 0 rz -180 deg; joints [0, 0, 0, 0, 0, 0]
  Call Extruder 0.7458
  MoveL (T3611) to (103.84, 121.16, 4.7) mm, rotated rx 180 ry 0 rz -180 deg; joints [0, 0, 0, 0, 0, 0]
  Call Extruder 0.10645
  MoveL (T3612) to (103.84, 117.66, 4.7) mm, rotated rx 180 ry 0 rz -180 deg; joints [0, 0, 0, 0, 0, 0]
  Call Extruder 0.15054
  MoveL (T3613) to (107.34, 121.16, 4.7) mm, rotated rx 180 ry 0 rz -180 deg; joints [0, 0, 0, 0, 0, 0]
  Call Extruder 0.03385
  MoveL (T3614) to (108.45, 121.16, 4.7) mm, rotated rx 180 ry 0 rz -180 deg; joints [0, 0, 0, 0, 0, 0]
  Call Extruder 0.46365
  MoveL (T3615) to (119.21, 110.39, 4.7) mm, rotated rx 180 ry 0 rz -180 deg; joints [0, 0, 0, 0, 0, 0]
  Call Extruder 0.01197
  MoveL (T3616) to (119.21, 110, 4.7) mm, rotated rx 180 ry 0 rz -180 deg; joints [0, 0, 0, 0, 0, 0]
  Call Extruder 0.18372
  MoveL (T3617) to (114.95, 105.74, 4.7) mm, rotated rx 180 ry 0 rz -180 deg; joints [0, 0, 0, 0, 0, 0]
  Call Extruder 0.00883
  MoveL (T3618) to (114.66, 105.74, 4.7) mm, rotated rx 180 ry 0 rz -180 deg; joints [0, 0, 0, 0, 0, 0]
  Call Extruder 0.46587
  MoveL (T3619) to (103.84, 116.55, 4.7) mm, rotated rx 180 ry 0 rz -180 deg; joints [0, 0, 0, 0, 0, 0]
  Call Extruder 0.07441
  MoveL (T3620) to (103.84, 114.11, 4.7) mm, rotated rx 180 ry 0 rz -180 deg; joints [0, 0, 0, 0, 0, 0]
  Set speed (45.0 mm/s)
  Call Extruder -1.6
  MoveL (T3621) to (103.84, 114.11, 4.7) mm, rotated rx 180 ry 0 rz -180 deg; joints [0, 0, 0, 0, 0, 0]
  Set speed (120.0 mm/s)
  MoveL (T3622) to (103.84, 114.11, 4.7) mm, rotated rx 180 ry 0 rz -180 deg; joints [0, 0, 0, 0, 0, 0]
  Call Extruder -0.38
  MoveL (T3623) to (103.84, 115.17, 4.7) mm, rotated rx 180 ry 0 rz -180 deg; joints [0, 0, 0, 0, 0, 0]
  Set speed (45.0 mm/s)
  Call Extruder -0.02
  MoveL (T3624) to (103.84, 115.17, 4.7) mm, rotated rx 180 ry 0 rz -180 deg; joints [0, 0, 0, 0, 0, 0]
  Set speed (150.0 mm/s)
  MoveL (T3625) to (103.84, 115.17, 6.7) mm, rotated rx 180 ry 0 rz -180 deg; joints [0, 0, 0, 0, 0, 0]
  MoveL (T3626) to (118.71, 121.16, 6.7) mm, rotated rx 180 ry 0 rz -180 deg; joints [0, 0, 0, 0, 0, 0]
  MoveL (T3627) to (118.71, 121.16, 4.7) mm, rotated rx 180 ry 0 rz -180 deg; joints [0, 0, 0, 0, 0, 0]
  Set speed (40.0 mm/s)
  Call Extruder 2.0
  MoveL (T3628) to (118.71, 121.16, 4.7) mm, rotated rx 180 ry 0 rz -180 deg; joints [0, 0, 0, 0, 0, 0]
  Set speed (26.7 mm/s)
  MoveL (T3629) to (118.71, 121.16, 4.7) mm, rotated rx 180 ry 0 rz -180 deg; joints [0, 0, 0, 0, 0, 0]
  Call Extruder 0.07441
  MoveL (T3630) to (121.16, 121.16, 4.7) mm, rotated rx 180 ry 0 rz -180 deg; joints [0, 0, 0, 0, 0, 0]
  Call Extruder 0.7458
  MoveL (T3631) to (103.84, 103.84, 4.7) mm, rotated rx 180 ry 0 rz -180 deg; joints [0, 0, 0, 0, 0, 0]
  Call Extruder 0.06976
  MoveL (T3632) to (106.13, 103.84, 4.7) mm, rotated rx 180 ry 0 rz -180 deg; joints [0, 0, 0, 0, 0, 0]
  Call Extruder 0.03667
  MoveL (T3633) to (106.14, 105.05, 4.7) mm, rotated rx 180 ry 0 rz -180 deg; joints [0, 0, 0, 0, 0, 0]
  Call Extruder 0.09868
  MoveL (T3634) to (103.84, 107.34, 4.7) mm, rotated rx 180 ry 0 rz -180 deg; joints [0, 0, 0, 0, 0, 0]
  Call Extruder 0.03385
  MoveL (T3635) to (103.84, 108.45, 4.7) mm, rotated rx 180 ry 0 rz -180 deg; joints [0, 0, 0, 0, 0, 0]
  Call Extruder 0.54738
  MoveL (T3636) to (116.55, 121.16, 4.7) mm, rotated rx 180 ry 0 rz -180 deg; joints [0, 0, 0, 0, 0, 0]
  Call Extruder 0.03385
  MoveL (T3637) to (117.66, 121.16, 4.7) mm, rotated rx 180 ry 0 rz -180 deg; joints [0, 0, 0, 0, 0, 0]
  Call Extruder 0.15054
  MoveL (T3638) to (121.16, 117.66, 4.7) mm, rotated rx 180 ry 0 rz -180 deg; joints [0, 0, 0, 0, 0, 0]
  Call Extruder 0.03385
  MoveL (T3639) to (121.16, 116.55, 4.7) mm, rotated rx 180 ry 0 rz -180 deg; joints [0, 0, 0, 0, 0, 0]
  Call Extruder 0.46587
  MoveL (T3640) to (110.34, 105.74, 4.7) mm, rotated rx 180 ry 0 rz -180 deg; joints [0, 0, 0, 0, 0, 0]
  Call Extruder 0.00883
  MoveL (T3641) to (110.05, 105.74, 4.7) mm, rotated rx 180 ry 0 rz -180 deg; joints [0, 0, 0, 0, 0, 0]
  Call Extruder 0.26745
  MoveL (T3642) to (103.84, 111.94, 4.7) mm, rotated rx 180 ry 0 rz -180 deg; joints [0, 0, 0, 0, 0, 0]
  Call Extruder 0.03385
  MoveL (T3643) to (103.84, 113.06, 4.7) mm, rotated rx 180 ry 0 rz -180 deg; joints [0, 0, 0, 0, 0, 0]
  Call Extruder 0.34896
  MoveL (T3644) to (111.94, 121.16, 4.7) mm, rotated rx 180 ry 0 rz -180 deg; joints [0, 0, 0, 0, 0, 0]
  Call Extruder 0.03385
  MoveL (T3645) to (113.06, 121.16, 4.7) mm, rotated rx 180 ry 0 rz -180 deg; joints [0, 0, 0, 0, 0, 0]
  Call Extruder 0.29344
  MoveL (T3646) to (119.87, 114.34, 4.7) mm, rotated rx 180 ry 0 rz -180 deg; joints [0, 0, 0, 0, 0, 0]
  Call Extruder 0.03926
  MoveL (T3647) to (121.16, 114.34, 4.7) mm, rotated rx 180 ry 0 rz -180 deg; joints [0, 0, 0, 0, 0, 0]
  Call Extruder 0.03515
  MoveL (T3648) to (121.16, 115.5, 4.7) mm, rotated rx 180 ry 0 rz -180 deg; joints [0, 0, 0, 0, 0, 0]
  Set speed (45.0 mm/s)
  Call Extruder -1.6
  MoveL (T3649) to (121.16, 115.5, 4.7) mm, rotated rx 180 ry 0 rz -180 deg; joints [0, 0, 0, 0, 0, 0]
  Set speed (120.0 mm/s)
  MoveL (T3650) to (121.16, 115.5, 4.7) mm, rotated rx 180 ry 0 rz -180 deg; joints [0, 0, 0, 0, 0, 0]
  Call Extruder -0.38
  MoveL (T3651) to (121.16, 114.43, 4.7) mm, rotated rx 180 ry 0 rz -180 deg; joints [0, 0, 0, 0, 0, 0]
  Set speed (45.0 mm/s)
  Call Extruder -0.02
  MoveL (T3652) to (121.16, 114.43, 4.7) mm, rotated rx 180 ry 0 rz -180 deg; joints [0, 0, 0, 0, 0, 0]
  Set speed (150.0 mm/s)
  MoveL (T3653) to (121.16, 114.43, 6.7) mm, rotated rx 180 ry 0 rz -180 deg; joints [0, 0, 0, 0, 0, 0]
  MoveL (T3654) to (104.34, 103.54, 6.7) mm, rotated rx 180 ry 0 rz -180 deg; joints [0, 0, 0, 0, 0, 0]
  MoveL (T3655) to (104.34, 103.54, 4.9) mm, rotated rx 180 ry 0 rz -180 deg; joints [0, 0, 0, 0, 0, 0]
  Set speed (40.0 mm/s)
  Call Extruder 2.0
  MoveL (T3656) to (104.34, 103.54, 4.9) mm, rotated rx 180 ry 0 rz -180 deg; joints [0, 0, 0, 0, 0, 0]
  Set speed (26.0 mm/s)
  MoveL (T3657) to (104.34, 103.54, 4.9) mm, rotated rx 180 ry 0 rz -180 deg; joints [0, 0, 0, 0, 0, 0]
  Call Extruder 0.0848
  MoveL (T3658) to (107.12, 103.54, 4.9) mm, rotated rx 180 ry 0 rz -180 deg; joints [0, 0, 0, 0, 0, 0]
  Call Extruder 0.05765
  MoveL (T3659) to (107.12, 105.43, 4.9) mm, rotated rx 180 ry 0 rz -180 deg; joints [0, 0, 0, 0, 0, 0]
  Call Extruder 0.11371
  MoveL (T3660) to (110.86, 105.43, 4.9) mm, rotated rx 180 ry 0 rz -180 deg; joints [0, 0, 0, 0, 0, 0]
  Call Extruder 0.05765
  MoveL (T3661) to (110.86, 103.54, 4.9) mm, rotated rx 180 ry 0 rz -180 deg; joints [0, 0, 0, 0, 0, 0]
  Call Extruder 0.07489
  MoveL (T3662) to (113.31, 103.54, 4.9) mm, rotated rx 180 ry 0 rz -180 deg; joints [0, 0, 0, 0, 0, 0]
  Call Extruder 0.05765
  MoveL (T3663) to (113.31, 105.43, 4.9) mm, rotated rx 180 ry 0 rz -180 deg; joints [0, 0, 0, 0, 0, 0]
  Call Extruder 0.1168
  MoveL (T3664) to (117.15, 105.43, 4.9) mm, rotated rx 180 ry 0 rz -180 deg; joints [0, 0, 0, 0, 0, 0]
  Call Extruder 0.05765
  MoveL (T3665) to (117.15, 103.54, 4.9) mm, rotated rx 180 ry 0 rz -180 deg; joints [0, 0, 0, 0, 0, 0]
  Call Extruder 0.13139
  MoveL (T3666) to (121.46, 103.54, 4.9) mm, rotated rx 180 ry 0 rz -180 deg; joints [0, 0, 0, 0, 0, 0]
  Call Extruder 0.20531
  MoveL (T3667) to (121.46, 110.28, 4.9) mm, rotated rx 180 ry 0 rz -180 deg; joints [0, 0, 0, 0, 0, 0]
  Call Extruder 0.0592
  MoveL (T3668) to (119.52, 110.28, 4.9) mm, rotated rx 180 ry 0 rz -180 deg; joints [0, 0, 0, 0, 0, 0]
  Call Extruder 0.11452
  MoveL (T3669) to (119.52, 114.04, 4.9) mm, rotated rx 180 ry 0 rz -180 deg; joints [0, 0, 0, 0, 0, 0]
  Call Extruder 0.05925
  MoveL (T3670) to (121.46, 114.04, 4.9) mm, rotated rx 180 ry 0 rz -180 deg; joints [0, 0, 0, 0, 0, 0]
  Call Extruder 0.22614
  MoveL (T3671) to (121.46, 121.46, 4.9) mm, rotated rx 180 ry 0 rz -180 deg; joints [0, 0, 0, 0, 0, 0]
  Call Extruder 0.54596
  MoveL (T3672) to (103.54, 121.46, 4.9) mm, rotated rx 180 ry 0 rz -180 deg; joints [0, 0, 0, 0, 0, 0]
  Call Extruder 0.54596
  MoveL (T3673) to (103.54, 103.54, 4.9) mm, rotated rx 180 ry 0 rz -180 deg; joints [0, 0, 0, 0, 0, 0]
  Call Extruder 0.02254
  MoveL (T3674) to (104.28, 103.54, 4.9) mm, rotated rx 180 ry 0 rz -180 deg; joints [0, 0, 0, 0, 0, 0]
  Set speed (150.0 mm/s)
  MoveL (T3675) to (103.53, 103.13, 4.9) mm, rotated rx 180 ry 0 rz -180 deg; joints [0, 0, 0, 0, 0, 0]
  Set speed (26.0 mm/s)
  MoveL (T3676) to (103.53, 103.13, 4.9) mm, rotated rx 180 ry 0 rz -180 deg; joints [0, 0, 0, 0, 0, 0]
  Call Extruder 0.12179
  MoveL (T3677) to (107.53, 103.13, 4.9) mm, rotated rx 180 ry 0 rz -180 deg; joints [0, 0, 0, 0, 0, 0]
  Call Extruder 0.05765
  MoveL (T3678) to (107.53, 105.02, 4.9) mm, rotated rx 180 ry 0 rz -180 deg; joints [0, 0, 0, 0, 0, 0]
  Call Extruder 0.08891
  MoveL (T3679) to (110.45, 105.02, 4.9) mm, rotated rx 180 ry 0 rz -180 deg; joints [0, 0, 0, 0, 0, 0]
  Call Extruder 0.05765
  MoveL (T3680) to (110.45, 103.13, 4.9) mm, rotated rx 180 ry 0 rz -180 deg; joints [0, 0, 0, 0, 0, 0]
  Call Extruder 0.0997
  MoveL (T3681) to (113.72, 103.13, 4.9) mm, rotated rx 180 ry 0 rz -180 deg; joints [0, 0, 0, 0, 0, 0]
  Call Extruder 0.05765
  MoveL (T3682) to (113.72, 105.02, 4.9) mm, rotated rx 180 ry 0 rz -180 deg; joints [0, 0, 0, 0, 0, 0]
  Call Extruder 0.09199
  MoveL (T3683) to (116.74, 105.02, 4.9) mm, rotated rx 180 ry 0 rz -180 deg; joints [0, 0, 0, 0, 0, 0]
  Call Extruder 0.05765
  MoveL (T3684) to (116.74, 103.13, 4.9) mm, rotated rx 180 ry 0 rz -180 deg; joints [0, 0, 0, 0, 0, 0]
  Call Extruder 0.15619
  MoveL (T3685) to (121.87, 103.13, 4.9) mm, rotated rx 180 ry 0 rz -180 deg; joints [0, 0, 0, 0, 0, 0]
  Call Extruder 0.23011
  MoveL (T3686) to (121.87, 110.69, 4.9) mm, rotated rx 180 ry 0 rz -180 deg; joints [0, 0, 0, 0, 0, 0]
  Call Extruder 0.05921
  MoveL (T3687) to (119.92, 110.69, 4.9) mm, rotated rx 180 ry 0 rz -180 deg; joints [0, 0, 0, 0, 0, 0]
  Call Extruder 0.08971
  MoveL (T3688) to (119.92, 113.63, 4.9) mm, rotated rx 180 ry 0 rz -180 deg; joints [0, 0, 0, 0, 0, 0]
  Call Extruder 0.05925
  MoveL (T3689) to (121.87, 113.63, 4.9) mm, rotated rx 180 ry 0 rz -180 deg; joints [0, 0, 0, 0, 0, 0]
  Call Extruder 0.25094
  MoveL (T3690) to (121.87, 121.87, 4.9) mm, rotated rx 180 ry 0 rz -180 deg; joints [0, 0, 0, 0, 0, 0]
  Call Extruder 0.57077
  MoveL (T3691) to (103.13, 121.87, 4.9) mm, rotated rx 180 ry 0 rz -180 deg; joints [0, 0, 0, 0, 0, 0]
  Call Extruder 0.57077
  MoveL (T3692) to (103.13, 103.13, 4.9) mm, rotated rx 180 ry 0 rz -180 deg; joints [0, 0, 0, 0, 0, 0]
  Call Extruder 0.01036
  MoveL (T3693) to (103.47, 103.13, 4.9) mm, rotated rx 180 ry 0 rz -180 deg; joints [0, 0, 0, 0, 0, 0]
  Set speed (150.0 mm/s)
  MoveL (T3694) to (102.72, 102.81, 4.9) mm, rotated rx 180 ry 0 rz -180 deg; joints [0, 0, 0, 0, 0, 0]
  Set speed (25.0 mm/s)
  MoveL (T3695) to (102.72, 102.81, 4.9) mm, rotated rx 180 ry 0 rz -180 deg; joints [0, 0, 0, 0, 0, 0]
  Call Extruder 0.00259
  MoveL (T3696) to (102.72, 102.72, 4.9) mm, rotated rx 180 ry 0 rz -180 deg; joints [0, 0, 0, 0, 0, 0]
  Call Extruder 0.15877
  MoveL (T3697) to (107.94, 102.72, 4.9) mm, rotated rx 180 ry 0 rz -180 deg; joints [0, 0, 0, 0, 0, 0]
  Call Extruder 0.05765
  MoveL (T3698) to (107.94, 104.62, 4.9) mm, rotated rx 180 ry 0 rz -180 deg; joints [0, 0, 0, 0, 0, 0]
  Call Extruder 0.06411
  MoveL (T3699) to (110.04, 104.62, 4.9) mm, rotated rx 180 ry 0 rz -180 deg; joints [0, 0, 0, 0, 0, 0]
  Call Extruder 0.05765
  MoveL (T3700) to (110.04, 102.72, 4.9) mm, rotated rx 180 ry 0 rz -180 deg; joints [0, 0, 0, 0, 0, 0]
  Call Extruder 0.12452
  MoveL (T3701) to (114.13, 102.72, 4.9) mm, rotated rx 180 ry 0 rz -180 deg; joints [0, 0, 0, 0, 0, 0]
  Call Extruder 0.05765
  MoveL (T3702) to (114.13, 104.62, 4.9) mm, rotated rx 180 ry 0 rz -180 deg; joints [0, 0, 0, 0, 0, 0]
  Call Extruder 0.06719
  MoveL (T3703) to (116.33, 104.62, 4.9) mm, rotated rx 180 ry 0 rz -180 deg; joints [0, 0, 0, 0, 0, 0]
  Call Extruder 0.05765
  MoveL (T3704) to (116.33, 102.72, 4.9) mm, rotated rx 180 ry 0 rz -180 deg; joints [0, 0, 0, 0, 0, 0]
  Call Extruder 0.18099
  MoveL (T3705) to (122.28, 102.72, 4.9) mm, rotated rx 180 ry 0 rz -180 deg; joints [0, 0, 0, 0, 0, 0]
  Call Extruder 0.25492
  MoveL (T3706) to (122.28, 111.09, 4.9) mm, rotated rx 180 ry 0 rz -180 deg; joints [0, 0, 0, 0, 0, 0]
  Call Extruder 0.05921
  MoveL (T3707) to (120.33, 111.09, 4.9) mm, rotated rx 180 ry 0 rz -180 deg; joints [0, 0, 0, 0, 0, 0]
  Call Extruder 0.06491
  MoveL (T3708) to (120.33, 113.22, 4.9) mm, rotated rx 180 ry 0 rz -180 deg; joints [0, 0, 0, 0, 0, 0]
  Call Extruder 0.05924
  MoveL (T3709) to (122.28, 113.22, 4.9) mm, rotated rx 180 ry 0 rz -180 deg; joints [0, 0, 0, 0, 0, 0]
  Call Extruder 0.27574
  MoveL (T3710) to (122.28, 122.28, 4.9) mm, rotated rx 180 ry 0 rz -180 deg; joints [0, 0, 0, 0, 0, 0]
  Call Extruder 0.59557
  MoveL (T3711) to (102.72, 122.28, 4.9) mm, rotated rx 180 ry 0 rz -180 deg; joints [0, 0, 0, 0, 0, 0]
  Call Extruder 0.59115
  MoveL (T3712) to (102.72, 102.87, 4.9) mm, rotated rx 180 ry 0 rz -180 deg; joints [0, 0, 0, 0, 0, 0]
  Set speed (150.0 mm/s)
  MoveL (T3713) to (102.78, 102.75, 4.9) mm, rotated rx 180 ry 0 rz -180 deg; joints [0, 0, 0, 0, 0, 0]
  Set speed (45.0 mm/s)
  Call Extruder -1.6
  MoveL (T3714) to (102.78, 102.75, 4.9) mm, rotated rx 180 ry 0 rz -180 deg; joints [0, 0, 0, 0, 0, 0]
  Set speed (120.0 mm/s)
  MoveL (T3715) to (102.78, 102.75, 4.9) mm, rotated rx 180 ry 0 rz -180 deg; joints [0, 0, 0, 0, 0, 0]
  Call Extruder -0.05166
  MoveL (T3716) to (102.72, 102.72, 4.9) mm, rotated rx 180 ry 0 rz -180 deg; joints [0, 0, 0, 0, 0, 0]
  Call Extruder -0.32834
  MoveL (T3717) to (103.65, 102.72, 4.9) mm, rotated rx 180 ry 0 rz -180 deg; joints [0, 0, 0, 0, 0, 0]
  Set speed (45.0 mm/s)
  Call Extruder -0.02
  MoveL (T3718) to (103.65, 102.72, 4.9) mm, rotated rx 180 ry 0 rz -180 deg; joints [0, 0, 0, 0, 0, 0]
  Set speed (150.0 mm/s)
  MoveL (T3719) to (103.65, 102.72, 6.9) mm, rotated rx 180 ry 0 rz -180 deg; joints [0, 0, 0, 0, 0, 0]
  MoveL (T3720) to (107, 104.69, 6.9) mm, rotated rx 180 ry 0 rz -180 deg; joints [0, 0, 0, 0, 0, 0]
  MoveL (T3721) to (107, 104.69, 4.9) mm, rotated rx 180 ry 0 rz -180 deg; joints [0, 0, 0, 0, 0, 0]
  Set speed (40.0 mm/s)
  Call Extruder 2.0
  MoveL (T3722) to (107, 104.69, 4.9) mm, rotated rx 180 ry 0 rz -180 deg; joints [0, 0, 0, 0, 0, 0]
  Set speed (26.0 mm/s)
  MoveL (T3723) to (107, 104.69, 4.9) mm, rotated rx 180 ry 0 rz -180 deg; joints [0, 0, 0, 0, 0, 0]
  Call Extruder 0.01596
  MoveL (T3724) to (106.65, 105.04, 4.9) mm, rotated rx 180 ry 0 rz -180 deg; joints [0, 0, 0, 0, 0, 0]
  Call Extruder 0.01983
  MoveL (T3725) to (106.65, 104.43, 4.9) mm, rotated rx 180 ry 0 rz -180 deg; joints [0, 0, 0, 0, 0, 0]
  Call Extruder 0.01596
  MoveL (T3726) to (107, 104.08, 4.9) mm, rotated rx 180 ry 0 rz -180 deg; joints [0, 0, 0, 0, 0, 0]
  Set speed (45.0 mm/s)
  Call Extruder -1.6
  MoveL (T3727) to (107, 104.08, 4.9) mm, rotated rx 180 ry 0 rz -180 deg; joints [0, 0, 0, 0, 0, 0]
  Set speed (120.0 mm/s)
  MoveL (T3728) to (107, 104.08, 4.9) mm, rotated rx 180 ry 0 rz -180 deg; joints [0, 0, 0, 0, 0, 0]
  Call Extruder -0.17547
  MoveL (T3729) to (106.65, 104.43, 4.9) mm, rotated rx 180 ry 0 rz -180 deg; joints [0, 0, 0, 0, 0, 0]
  Call Extruder -0.20453
  MoveL (T3730) to (106.65, 105, 4.9) mm, rotated rx 180 ry 0 rz -180 deg; joints [0, 0, 0, 0, 0, 0]
  Set speed (45.0 mm/s)
  Call Extruder -0.02
  MoveL (T3731) to (106.65, 105, 4.9) mm, rotated rx 180 ry 0 rz -180 deg; joints [0, 0, 0, 0, 0, 0]
  Set speed (150.0 mm/s)
  MoveL (T3732) to (106.65, 105, 6.9) mm, rotated rx 180 ry 0 rz -180 deg; joints [0, 0, 0, 0, 0, 0]
  MoveL (T3733) to (111.28, 105.64, 6.9) mm, rotated rx 180 ry 0 rz -180 deg; joints [0, 0, 0, 0, 0, 0]
  MoveL (T3734) to (111.28, 105.64, 4.9) mm, rotated rx 180 ry 0 rz -180 deg; joints [0, 0, 0, 0, 0, 0]
  Set speed (40.0 mm/s)
  Call Extruder 2.0
  MoveL (T3735) to (111.28, 105.64, 4.9) mm, rotated rx 180 ry 0 rz -180 deg; joints [0, 0, 0, 0, 0, 0]
  Set speed (26.0 mm/s)
  MoveL (T3736) to (111.28, 105.64, 4.9) mm, rotated rx 180 ry 0 rz -180 deg; joints [0, 0, 0, 0, 0, 0]
  Call Extruder 0.01539
  MoveL (T3737) to (111.59, 105.33, 4.9) mm, rotated rx 180 ry 0 rz -180 deg; joints [0, 0, 0, 0, 0, 0]
  Call Extruder 0.02341
  MoveL (T3738) to (111.59, 104.67, 4.9) mm, rotated rx 180 ry 0 rz -180 deg; joints [0, 0, 0, 0, 0, 0]
  Call Extruder 0.0215
  MoveL (T3739) to (111.16, 105.1, 4.9) mm, rotated rx 180 ry 0 rz -180 deg; joints [0, 0, 0, 0, 0, 0]
  Call Extruder 0.02341
  MoveL (T3740) to (111.16, 104.44, 4.9) mm, rotated rx 180 ry 0 rz -180 deg; joints [0, 0, 0, 0, 0, 0]
  Call Extruder 0.03062
  MoveL (T3741) to (111.78, 103.82, 4.9) mm, rotated rx 180 ry 0 rz -180 deg; joints [0, 0, 0, 0, 0, 0]
  Set speed (45.0 mm/s)
  Call Extruder -1.6
  MoveL (T3742) to (111.78, 103.82, 4.9) mm, rotated rx 180 ry 0 rz -180 deg; joints [0, 0, 0, 0, 0, 0]
  Set speed (120.0 mm/s)
  MoveL (T3743) to (111.78, 103.82, 4.9) mm, rotated rx 180 ry 0 rz -180 deg; joints [0, 0, 0, 0, 0, 0]
  Call Extruder -0.30984
  MoveL (T3744) to (111.16, 104.44, 4.9) mm, rotated rx 180 ry 0 rz -180 deg; joints [0, 0, 0, 0, 0, 0]
  Call Extruder -0.07016
  MoveL (T3745) to (111.16, 104.63, 4.9) mm, rotated rx 180 ry 0 rz -180 deg; joints [0, 0, 0, 0, 0, 0]
  Set speed (45.0 mm/s)
  Call Extruder -0.02
  MoveL (T3746) to (111.16, 104.63, 4.9) mm, rotated rx 180 ry 0 rz -180 deg; joints [0, 0, 0, 0, 0, 0]
  Set speed (150.0 mm/s)
  MoveL (T3747) to (111.16, 104.63, 6.9) mm, rotated rx 180 ry 0 rz -180 deg; joints [0, 0, 0, 0, 0, 0]
  MoveL (T3748) to (113.19, 105.27, 6.9) mm, rotated rx 180 ry 0 rz -180 deg; joints [0, 0, 0, 0, 0, 0]
  MoveL (T3749) to (113.19, 105.27, 4.9) mm, rotated rx 180 ry 0 rz -180 deg; joints [0, 0, 0, 0, 0, 0]
  Set speed (40.0 mm/s)
  Call Extruder 2.0
  MoveL (T3750) to (113.19, 105.27, 4.9) mm, rotated rx 180 ry 0 rz -180 deg; joints [0, 0, 0, 0, 0, 0]
  Set speed (26.0 mm/s)
  MoveL (T3751) to (113.19, 105.27, 4.9) mm, rotated rx 180 ry 0 rz -180 deg; joints [0, 0, 0, 0, 0, 0]
  Call Extruder 0.00974
  MoveL (T3752) to (113, 105.46, 4.9) mm, rotated rx 180 ry 0 rz -180 deg; joints [0, 0, 0, 0, 0, 0]
  Call Extruder 0.01318
  MoveL (T3753) to (112.64, 105.46, 4.9) mm, rotated rx 180 ry 0 rz -180 deg; joints [0, 0, 0, 0, 0, 0]
  Call Extruder 0.00415
  MoveL (T3754) to (112.56, 105.38, 4.9) mm, rotated rx 180 ry 0 rz -180 deg; joints [0, 0, 0, 0, 0, 0]
  Call Extruder 0.00571
  MoveL (T3755) to (112.56, 105.22, 4.9) mm, rotated rx 180 ry 0 rz -180 deg; joints [0, 0, 0, 0, 0, 0]
  Call Extruder 0.02316
  MoveL (T3756) to (113.01, 104.77, 4.9) mm, rotated rx 180 ry 0 rz -180 deg; joints [0, 0, 0, 0, 0, 0]
  Call Extruder 0.02477
  MoveL (T3757) to (113.01, 104.08, 4.9) mm, rotated rx 180 ry 0 rz -180 deg; joints [0, 0, 0, 0, 0, 0]
  Call Extruder 0.02316
  MoveL (T3758) to (112.56, 104.54, 4.9) mm, rotated rx 180 ry 0 rz -180 deg; joints [0, 0, 0, 0, 0, 0]
  Call Extruder 0.02477
  MoveL (T3759) to (112.56, 103.85, 4.9) mm, rotated rx 180 ry 0 rz -180 deg; joints [0, 0, 0, 0, 0, 0]
  Call Extruder 0.00973
  MoveL (T3760) to (112.75, 103.66, 4.9) mm, rotated rx 180 ry 0 rz -180 deg; joints [0, 0, 0, 0, 0, 0]
  Set speed (45.0 mm/s)
  Call Extruder -1.6
  MoveL (T3761) to (112.75, 103.66, 4.9) mm, rotated rx 180 ry 0 rz -180 deg; joints [0, 0, 0, 0, 0, 0]
  Set speed (120.0 mm/s)
  MoveL (T3762) to (112.75, 103.66, 4.9) mm, rotated rx 180 ry 0 rz -180 deg; joints [0, 0, 0, 0, 0, 0]
  Call Extruder -0.09575
  MoveL (T3763) to (112.56, 103.85, 4.9) mm, rotated rx 180 ry 0 rz -180 deg; joints [0, 0, 0, 0, 0, 0]
  Call Extruder -0.24379
  MoveL (T3764) to (112.56, 104.54, 4.9) mm, rotated rx 180 ry 0 rz -180 deg; joints [0, 0, 0, 0, 0, 0]
  Call Extruder -0.04045
  MoveL (T3765) to (112.64, 104.45, 4.9) mm, rotated rx 180 ry 0 rz -180 deg; joints [0, 0, 0, 0, 0, 0]
  Set speed (45.0 mm/s)
  Call Extruder -0.02
  MoveL (T3766) to (112.64, 104.45, 4.9) mm, rotated rx 180 ry 0 rz -180 deg; joints [0, 0, 0, 0, 0, 0]
  Set speed (150.0 mm/s)
  MoveL (T3767) to (112.64, 104.45, 6.9) mm, rotated rx 180 ry 0 rz -180 deg; joints [0, 0, 0, 0, 0, 0]
  MoveL (T3768) to (117.4, 105.64, 6.9) mm, rotated rx 180 ry 0 rz -180 deg; joints [0, 0, 0, 0, 0, 0]
  MoveL (T3769) to (117.4, 105.64, 4.9) mm, rotated rx 180 ry 0 rz -180 deg; joints [0, 0, 0, 0, 0, 0]
  Set speed (40.0 mm/s)
  Call Extruder 2.0
  MoveL (T3770) to (117.4, 105.64, 4.9) mm, rotated rx 180 ry 0 rz -180 deg; joints [0, 0, 0, 0, 0, 0]
  Set speed (26.0 mm/s)
  MoveL (T3771) to (117.4, 105.64, 4.9) mm, rotated rx 180 ry 0 rz -180 deg; joints [0, 0, 0, 0, 0, 0]
  Call Extruder 0.013
  MoveL (T3772) to (117.68, 105.36, 4.9) mm, rotated rx 180 ry 0 rz -180 deg; joints [0, 0, 0, 0, 0, 0]
  Call Extruder 0.01991
  MoveL (T3773) to (117.68, 104.74, 4.9) mm, rotated rx 180 ry 0 rz -180 deg; joints [0, 0, 0, 0, 0, 0]
  Call Extruder 0.01042
  MoveL (T3774) to (117.45, 104.97, 4.9) mm, rotated rx 180 ry 0 rz -180 deg; joints [0, 0, 0, 0, 0, 0]
  Call Extruder 0.01991
  MoveL (T3775) to (117.45, 104.36, 4.9) mm, rotated rx 180 ry 0 rz -180 deg; joints [0, 0, 0, 0, 0, 0]
  Call Extruder 0.01883
  MoveL (T3776) to (117.86, 103.95, 4.9) mm, rotated rx 180 ry 0 rz -180 deg; joints [0, 0, 0, 0, 0, 0]
  Set speed (45.0 mm/s)
  Call Extruder -1.6
  MoveL (T3777) to (117.86, 103.95, 4.9) mm, rotated rx 180 ry 0 rz -180 deg; joints [0, 0, 0, 0, 0, 0]
  Set speed (120.0 mm/s)
  MoveL (T3778) to (117.86, 103.95, 4.9) mm, rotated rx 180 ry 0 rz -180 deg; joints [0, 0, 0, 0, 0, 0]
  Call Extruder -0.20676
  MoveL (T3779) to (117.45, 104.36, 4.9) mm, rotated rx 180 ry 0 rz -180 deg; joints [0, 0, 0, 0, 0, 0]
  Call Extruder -0.17324
  MoveL (T3780) to (117.45, 104.84, 4.9) mm, rotated rx 180 ry 0 rz -180 deg; joints [0, 0, 0, 0, 0, 0]
  Set speed (45.0 mm/s)
  Call Extruder -0.02
  MoveL (T3781) to (117.45, 104.84, 4.9) mm, rotated rx 180 ry 0 rz -180 deg; joints [0, 0, 0, 0, 0, 0]
  Set speed (150.0 mm/s)
  MoveL (T3782) to (117.45, 104.84, 6.9) mm, rotated rx 180 ry 0 rz -180 deg; joints [0, 0, 0, 0, 0, 0]
  MoveL (T3783) to (121.16, 109.05, 6.9) mm, rotated rx 180 ry 0 rz -180 deg; joints [0, 0, 0, 0, 0, 0]
  MoveL (T3784) to (121.16, 109.05, 4.9) mm, rotated rx 180 ry 0 rz -180 deg; joints [0, 0, 0, 0, 0, 0]
  Set speed (40.0 mm/s)
  Call Extruder 2.0
  MoveL (T3785) to (121.16, 109.05, 4.9) mm, rotated rx 180 ry 0 rz -180 deg; joints [0, 0, 0, 0, 0, 0]
  Set speed (26.0 mm/s)
  MoveL (T3786) to (121.16, 109.05, 4.9) mm, rotated rx 180 ry 0 rz -180 deg; joints [0, 0, 0, 0, 0, 0]
  Call Extruder 0.02803
  MoveL (T3787) to (121.16, 109.97, 4.9) mm, rotated rx 180 ry 0 rz -180 deg; joints [0, 0, 0, 0, 0, 0]
  Call Extruder 0.04638
  MoveL (T3788) to (119.63, 109.97, 4.9) mm, rotated rx 180 ry 0 rz -180 deg; joints [0, 0, 0, 0, 0, 0]
  Call Extruder 0.06559
  MoveL (T3789) to (121.16, 108.45, 4.9) mm, rotated rx 180 ry 0 rz -180 deg; joints [0, 0, 0, 0, 0, 0]
  Call Extruder 0.03385
  MoveL (T3790) to (121.16, 107.34, 4.9) mm, rotated rx 180 ry 0 rz -180 deg; joints [0, 0, 0, 0, 0, 0]
  Call Extruder 0.13221
  MoveL (T3791) to (118.09, 104.27, 4.9) mm, rotated rx 180 ry 0 rz -180 deg; joints [0, 0, 0, 0, 0, 0]
  Call Extruder 0.01296
  MoveL (T3792) to (118.09, 103.84, 4.9) mm, rotated rx 180 ry 0 rz -180 deg; joints [0, 0, 0, 0, 0, 0]
  Call Extruder 0.09348
  MoveL (T3793) to (121.16, 103.84, 4.9) mm, rotated rx 180 ry 0 rz -180 deg; joints [0, 0, 0, 0, 0, 0]
  Call Extruder 0.7458
  MoveL (T3794) to (103.84, 121.16, 4.9) mm, rotated rx 180 ry 0 rz -180 deg; joints [0, 0, 0, 0, 0, 0]
  Call Extruder 0.10645
  MoveL (T3795) to (103.84, 117.66, 4.9) mm, rotated rx 180 ry 0 rz -180 deg; joints [0, 0, 0, 0, 0, 0]
  Call Extruder 0.15054
  MoveL (T3796) to (107.34, 121.16, 4.9) mm, rotated rx 180 ry 0 rz -180 deg; joints [0, 0, 0, 0, 0, 0]
  Call Extruder 0.03385
  MoveL (T3797) to (108.45, 121.16, 4.9) mm, rotated rx 180 ry 0 rz -180 deg; joints [0, 0, 0, 0, 0, 0]
  Call Extruder 0.46366
  MoveL (T3798) to (119.21, 110.39, 4.9) mm, rotated rx 180 ry 0 rz -180 deg; joints [0, 0, 0, 0, 0, 0]
  Call Extruder 0.01195
  MoveL (T3799) to (119.21, 110, 4.9) mm, rotated rx 180 ry 0 rz -180 deg; joints [0, 0, 0, 0, 0, 0]
  Call Extruder 0.18372
  MoveL (T3800) to (114.95, 105.74, 4.9) mm, rotated rx 180 ry 0 rz -180 deg; joints [0, 0, 0, 0, 0, 0]
  Call Extruder 0.00884
  MoveL (T3801) to (114.66, 105.74, 4.9) mm, rotated rx 180 ry 0 rz -180 deg; joints [0, 0, 0, 0, 0, 0]
  Call Extruder 0.46586
  MoveL (T3802) to (103.84, 116.55, 4.9) mm, rotated rx 180 ry 0 rz -180 deg; joints [0, 0, 0, 0, 0, 0]
  Call Extruder 0.07441
  MoveL (T3803) to (103.84, 114.11, 4.9) mm, rotated rx 180 ry 0 rz -180 deg; joints [0, 0, 0, 0, 0, 0]
  Set speed (45.0 mm/s)
  Call Extruder -1.6
  MoveL (T3804) to (103.84, 114.11, 4.9) mm, rotated rx 180 ry 0 rz -180 deg; joints [0, 0, 0, 0, 0, 0]
  Set speed (120.0 mm/s)
  MoveL (T3805) to (103.84, 114.11, 4.9) mm, rotated rx 180 ry 0 rz -180 deg; joints [0, 0, 0, 0, 0, 0]
  Call Extruder -0.38
  MoveL (T3806) to (103.84, 115.17, 4.9) mm, rotated rx 180 ry 0 rz -180 deg; joints [0, 0, 0, 0, 0, 0]
  Set speed (45.0 mm/s)
  Call Extruder -0.02
  MoveL (T3807) to (103.84, 115.17, 4.9) mm, rotated rx 180 ry 0 rz -180 deg; joints [0, 0, 0, 0, 0, 0]
  Set speed (150.0 mm/s)
  MoveL (T3808) to (103.84, 115.17, 6.9) mm, rotated rx 180 ry 0 rz -180 deg; joints [0, 0, 0, 0, 0, 0]
  MoveL (T3809) to (118.71, 121.16, 6.9) mm, rotated rx 180 ry 0 rz -180 deg; joints [0, 0, 0, 0, 0, 0]
  MoveL (T3810) to (118.71, 121.16, 4.9) mm, rotated rx 180 ry 0 rz -180 deg; joints [0, 0, 0, 0, 0, 0]
  Set speed (40.0 mm/s)
  Call Extruder 2.0
  MoveL (T3811) to (118.71, 121.16, 4.9) mm, rotated rx 180 ry 0 rz -180 deg; joints [0, 0, 0, 0, 0, 0]
  Set speed (26.0 mm/s)
  MoveL (T3812) to (118.71, 121.16, 4.9) mm, rotated rx 180 ry 0 rz -180 deg; joints [0, 0, 0, 0, 0, 0]
  Call Extruder 0.07441
  MoveL (T3813) to (121.16, 121.16, 4.9) mm, rotated rx 180 ry 0 rz -180 deg; joints [0, 0, 0, 0, 0, 0]
  Call Extruder 0.7458
  MoveL (T3814) to (103.84, 103.84, 4.9) mm, rotated rx 180 ry 0 rz -180 deg; joints [0, 0, 0, 0, 0, 0]
  Call Extruder 0.07314
  MoveL (T3815) to (106.25, 103.84, 4.9) mm, rotated rx 180 ry 0 rz -180 deg; joints [0, 0, 0, 0, 0, 0]
  Call Extruder 0.03329
  MoveL (T3816) to (106.25, 104.94, 4.9) mm, rotated rx 180 ry 0 rz -180 deg; joints [0, 0, 0, 0, 0, 0]
  Call Extruder 0.10346
  MoveL (T3817) to (103.84, 107.34, 4.9) mm, rotated rx 180 ry 0 rz -180 deg; joints [0, 0, 0, 0, 0, 0]
  Call Extruder 0.03385
  MoveL (T3818) to (103.84, 108.45, 4.9) mm, rotated rx 180 ry 0 rz -180 deg; joints [0, 0, 0, 0, 0, 0]
  Call Extruder 0.54738
  MoveL (T3819) to (116.55, 121.16, 4.9) mm, rotated rx 180 ry 0 rz -180 deg; joints [0, 0, 0, 0, 0, 0]
  Call Extruder 0.03385
  MoveL (T3820) to (117.66, 121.16, 4.9) mm, rotated rx 180 ry 0 rz -180 deg; joints [0, 0, 0, 0, 0, 0]
  Call Extruder 0.15054
  MoveL (T3821) to (121.16, 117.66, 4.9) mm, rotated rx 180 ry 0 rz -180 deg; joints [0, 0, 0, 0, 0, 0]
  Call Extruder 0.03385
  MoveL (T3822) to (121.16, 116.55, 4.9) mm, rotated rx 180 ry 0 rz -180 deg; joints [0, 0, 0, 0, 0, 0]
  Call Extruder 0.46586
  MoveL (T3823) to (110.34, 105.74, 4.9) mm, rotated rx 180 ry 0 rz -180 deg; joints [0, 0, 0, 0, 0, 0]
  Call Extruder 0.00884
  MoveL (T3824) to (110.05, 105.74, 4.9) mm, rotated rx 180 ry 0 rz -180 deg; joints [0, 0, 0, 0, 0, 0]
  Call Extruder 0.26744
  MoveL (T3825) to (103.84, 111.94, 4.9) mm, rotated rx 180 ry 0 rz -180 deg; joints [0, 0, 0, 0, 0, 0]
  Call Extruder 0.03385
  MoveL (T3826) to (103.84, 113.06, 4.9) mm, rotated rx 180 ry 0 rz -180 deg; joints [0, 0, 0, 0, 0, 0]
  Call Extruder 0.34896
  MoveL (T3827) to (111.94, 121.16, 4.9) mm, rotated rx 180 ry 0 rz -180 deg; joints [0, 0, 0, 0, 0, 0]
  Call Extruder 0.03385
  MoveL (T3828) to (113.06, 121.16, 4.9) mm, rotated rx 180 ry 0 rz -180 deg; joints [0, 0, 0, 0, 0, 0]
  Call Extruder 0.29353
  MoveL (T3829) to (119.87, 114.34, 4.9) mm, rotated rx 180 ry 0 rz -180 deg; joints [0, 0, 0, 0, 0, 0]
  Call Extruder 0.03919
  MoveL (T3830) to (121.16, 114.34, 4.9) mm, rotated rx 180 ry 0 rz -180 deg; joints [0, 0, 0, 0, 0, 0]
  Call Extruder 0.03521
  MoveL (T3831) to (121.16, 115.5, 4.9) mm, rotated rx 180 ry 0 rz -180 deg; joints [0, 0, 0, 0, 0, 0]
  Set speed (45.0 mm/s)
  Call Extruder -1.6
  MoveL (T3832) to (121.16, 115.5, 4.9) mm, rotated rx 180 ry 0 rz -180 deg; joints [0, 0, 0, 0, 0, 0]
  Set speed (120.0 mm/s)
  MoveL (T3833) to (121.16, 115.5, 4.9) mm, rotated rx 180 ry 0 rz -180 deg; joints [0, 0, 0, 0, 0, 0]
  Call Extruder -0.38
  MoveL (T3834) to (121.16, 114.43, 4.9) mm, rotated rx 180 ry 0 rz -180 deg; joints [0, 0, 0, 0, 0, 0]
  Set speed (45.0 mm/s)
  Call Extruder -0.02
  MoveL (T3835) to (121.16, 114.43, 4.9) mm, rotated rx 180 ry 0 rz -180 deg; joints [0, 0, 0, 0, 0, 0]
  Set speed (150.0 mm/s)
  MoveL (T3836) to (121.16, 114.43, 6.9) mm, rotated rx 180 ry 0 rz -180 deg; joints [0, 0, 0, 0, 0, 0]
  MoveL (T3837) to (104.34, 103.54, 6.9) mm, rotated rx 180 ry 0 rz -180 deg; joints [0, 0, 0, 0, 0, 0]
  MoveL (T3838) to (104.34, 103.54, 5.1) mm, rotated rx 180 ry 0 rz -180 deg; joints [0, 0, 0, 0, 0, 0]
  Set speed (40.0 mm/s)
  Call Extruder 2.0
  MoveL (T3839) to (104.34, 103.54, 5.1) mm, rotated rx 180 ry 0 rz -180 deg; joints [0, 0, 0, 0, 0, 0]
  Set speed (25.7 mm/s)
  MoveL (T3840) to (104.34, 103.54, 5.1) mm, rotated rx 180 ry 0 rz -180 deg; joints [0, 0, 0, 0, 0, 0]
  Call Extruder 0.08819
  MoveL (T3841) to (107.23, 103.54, 5.1) mm, rotated rx 180 ry 0 rz -180 deg; joints [0, 0, 0, 0, 0, 0]
  Call Extruder 0.05765
  MoveL (T3842) to (107.23, 105.43, 5.1) mm, rotated rx 180 ry 0 rz -180 deg; joints [0, 0, 0, 0, 0, 0]
  Call Extruder 0.11394
  MoveL (T3843) to (110.97, 105.43, 5.1) mm, rotated rx 180 ry 0 rz -180 deg; joints [0, 0, 0, 0, 0, 0]
  Call Extruder 0.05765
  MoveL (T3844) to (110.97, 103.54, 5.1) mm, rotated rx 180 ry 0 rz -180 deg; joints [0, 0, 0, 0, 0, 0]
  Call Extruder 0.06757
  MoveL (T3845) to (113.19, 103.54, 5.1) mm, rotated rx 180 ry 0 rz -180 deg; joints [0, 0, 0, 0, 0, 0]
  Call Extruder 0.05765
  MoveL (T3846) to (113.19, 105.43, 5.1) mm, rotated rx 180 ry 0 rz -180 deg; joints [0, 0, 0, 0, 0, 0]
  Call Extruder 0.11666
  MoveL (T3847) to (117.02, 105.43, 5.1) mm, rotated rx 180 ry 0 rz -180 deg; joints [0, 0, 0, 0, 0, 0]
  Call Extruder 0.05765
  MoveL (T3848) to (117.02, 103.54, 5.1) mm, rotated rx 180 ry 0 rz -180 deg; joints [0, 0, 0, 0, 0, 0]
  Call Extruder 0.13525
  MoveL (T3849) to (121.46, 103.54, 5.1) mm, rotated rx 180 ry 0 rz -180 deg; joints [0, 0, 0, 0, 0, 0]
  Call Extruder 0.20524
  MoveL (T3850) to (121.46, 110.28, 5.1) mm, rotated rx 180 ry 0 rz -180 deg; joints [0, 0, 0, 0, 0, 0]
  Call Extruder 0.05919
  MoveL (T3851) to (119.52, 110.28, 5.1) mm, rotated rx 180 ry 0 rz -180 deg; joints [0, 0, 0, 0, 0, 0]
  Call Extruder 0.11452
  MoveL (T3852) to (119.52, 114.03, 5.1) mm, rotated rx 180 ry 0 rz -180 deg; joints [0, 0, 0, 0, 0, 0]
  Call Extruder 0.05924
  MoveL (T3853) to (121.46, 114.03, 5.1) mm, rotated rx 180 ry 0 rz -180 deg; joints [0, 0, 0, 0, 0, 0]
  Call Extruder 0.22621
  MoveL (T3854) to (121.46, 121.46, 5.1) mm, rotated rx 180 ry 0 rz -180 deg; joints [0, 0, 0, 0, 0, 0]
  Call Extruder 0.54596
  MoveL (T3855) to (103.54, 121.46, 5.1) mm, rotated rx 180 ry 0 rz -180 deg; joints [0, 0, 0, 0, 0, 0]
  Call Extruder 0.54596
  MoveL (T3856) to (103.54, 103.54, 5.1) mm, rotated rx 180 ry 0 rz -180 deg; joints [0, 0, 0, 0, 0, 0]
  Call Extruder 0.02254
  MoveL (T3857) to (104.28, 103.54, 5.1) mm, rotated rx 180 ry 0 rz -180 deg; joints [0, 0, 0, 0, 0, 0]
  Set speed (150.0 mm/s)
  MoveL (T3858) to (103.53, 103.13, 5.1) mm, rotated rx 180 ry 0 rz -180 deg; joints [0, 0, 0, 0, 0, 0]
  Set speed (25.7 mm/s)
  MoveL (T3859) to (103.53, 103.13, 5.1) mm, rotated rx 180 ry 0 rz -180 deg; joints [0, 0, 0, 0, 0, 0]
  Call Extruder 0.12517
  MoveL (T3860) to (107.64, 103.13, 5.1) mm, rotated rx 180 ry 0 rz -180 deg; joints [0, 0, 0, 0, 0, 0]
  Call Extruder 0.05765
  MoveL (T3861) to (107.64, 105.03, 5.1) mm, rotated rx 180 ry 0 rz -180 deg; joints [0, 0, 0, 0, 0, 0]
  Call Extruder 0.08914
  MoveL (T3862) to (110.57, 105.03, 5.1) mm, rotated rx 180 ry 0 rz -180 deg; joints [0, 0, 0, 0, 0, 0]
  Call Extruder 0.05765
  MoveL (T3863) to (110.57, 103.13, 5.1) mm, rotated rx 180 ry 0 rz -180 deg; joints [0, 0, 0, 0, 0, 0]
  Call Extruder 0.09238
  MoveL (T3864) to (113.6, 103.13, 5.1) mm, rotated rx 180 ry 0 rz -180 deg; joints [0, 0, 0, 0, 0, 0]
  Call Extruder 0.05765
  MoveL (T3865) to (113.6, 105.03, 5.1) mm, rotated rx 180 ry 0 rz -180 deg; joints [0, 0, 0, 0, 0, 0]
  Call Extruder 0.09185
  MoveL (T3866) to (116.61, 105.03, 5.1) mm, rotated rx 180 ry 0 rz -180 deg; joints [0, 0, 0, 0, 0, 0]
  Call Extruder 0.05765
  MoveL (T3867) to (116.61, 103.13, 5.1) mm, rotated rx 180 ry 0 rz -180 deg; joints [0, 0, 0, 0, 0, 0]
  Call Extruder 0.16004
  MoveL (T3868) to (121.87, 103.13, 5.1) mm, rotated rx 180 ry 0 rz -180 deg; joints [0, 0, 0, 0, 0, 0]
  Call Extruder 0.23005
  MoveL (T3869) to (121.87, 110.68, 5.1) mm, rotated rx 180 ry 0 rz -180 deg; joints [0, 0, 0, 0, 0, 0]
  Call Extruder 0.0592
  MoveL (T3870) to (119.92, 110.68, 5.1) mm, rotated rx 180 ry 0 rz -180 deg; joints [0, 0, 0, 0, 0, 0]
  Call Extruder 0.08971
  MoveL (T3871) to (119.92, 113.63, 5.1) mm, rotated rx 180 ry 0 rz -180 deg; joints [0, 0, 0, 0, 0, 0]
  Call Extruder 0.05924
  MoveL (T3872) to (121.87, 113.63, 5.1) mm, rotated rx 180 ry 0 rz -180 deg; joints [0, 0, 0, 0, 0, 0]
  Call Extruder 0.251
  MoveL (T3873) to (121.87, 121.87, 5.1) mm, rotated rx 180 ry 0 rz -180 deg; joints [0, 0, 0, 0, 0, 0]
  Call Extruder 0.57077
